LIN {X 0,Y 467.641,Z 718.232,A -85,B 0,C 180,E1 -7755.695,E2 -7755.695} C_VEL
LIN {X 0,Y 467.624,Z 718.234,A -85,B 0,C 180,E1 -7759.308,E2 -7759.308} C_VEL
LIN {X 0,Y 467.537,Z 718.247,A -85,B 0,C 180,E1 -7762.074,E2 -7762.074} C_VEL
LIN {X 0,Y 467.557,Z 718.246,A -85,B 0,C 180,E1 -7764.89,E2 -7764.89} C_VEL
LIN {X 0,Y 467.58,Z 718.239,A -85,B 0,C 180,E1 -7767.772,E2 -7767.772} C_VEL
LIN {X 0,Y 467.569,Z 718.244,A -85,B 0,C 180,E1 -7771.045,E2 -7771.045} C_VEL
LIN {X 0,Y 467.578,Z 718.242,A -85,B 0,C 180,E1 -7774.24,E2 -7774.24} C_VEL
LIN {X 0,Y 467.537,Z 718.248,A -85,B 0,C 180,E1 -7777.184,E2 -7777.184} C_VEL
LIN {X 0,Y 467.558,Z 718.244,A -85,B 0,C 180,E1 -7780.267,E2 -7780.267} C_VEL
LIN {X 0,Y 467.546,Z 718.243,A -85,B 0,C 180,E1 -7783.746,E2 -7783.746} C_VEL
LIN {X 0,Y 467.546,Z 718.244,A -85,B 0,C 180,E1 -7786.254,E2 -7786.254} C_VEL
LIN {X 0,Y 467.558,Z 718.242,A -85,B 0,C 180,E1 -7789.733,E2 -7789.733} C_VEL
LIN {X 0,Y 467.519,Z 718.25,A -85,B 0,C 180,E1 -7792.819,E2 -7792.819} C_VEL
LIN {X 0,Y 467.566,Z 718.242,A -85,B 0,C 180,E1 -7795.762,E2 -7795.762} C_VEL
LIN {X 0,Y 467.537,Z 718.248,A -85,B 0,C 180,E1 -7798.962,E2 -7798.962} C_VEL
LIN {X 0,Y 467.543,Z 718.244,A -85,B 0,C 180,E1 -7802.226,E2 -7802.226} C_VEL
LIN {X 0,Y 467.551,Z 718.246,A -85,B 0,C 180,E1 -7805.11,E2 -7805.11} C_VEL
LIN {X 0,Y 467.534,Z 718.246,A -85,B 0,C 180,E1 -7807.926,E2 -7807.926} C_VEL
LIN {X 0,Y 467.623,Z 718.234,A -85,B 0,C 180,E1 -7810.692,E2 -7810.692} C_VEL
LIN {X 0,Y 467.64,Z 718.231,A -85,B 0,C 180,E1 -7814.305,E2 -7814.305} C_VEL
LIN {X 0,Y 467.591,Z 718.24,A -85,B 0,C 180,E1 -7815.403,E2 -7815.403} C_VEL
LIN {X 0,Y 466.918,Z 718.323,A -85,B 0,C 180,E1 -7816.122,E2 -7816.122} C_VEL
LIN {X 0,Y 464.072,Z 718.68,A -85,B 0,C 180,E1 -7817.291,E2 -7817.291} C_VEL
LIN {X 0,Y 461.669,Z 718.976,A -85,B 0,C 180,E1 -7818.233,E2 -7818.233} C_VEL
LIN {X 0,Y 460.636,Z 719.106,A -85,B 0,C 180,E1 -7818.961,E2 -7818.961} C_VEL
LIN {X 0,Y 460.55,Z 719.116,A -85,B 0,C 180,E1 -7819.207,E2 -7819.207} C_VEL
LIN {X 0,Y 460.666,Z 719.1,A -85,B 0,C 180,E1 -7822.594,E2 -7822.594} C_VEL
LIN {X 0,Y 460.676,Z 719.099,A -85,B 0,C 180,E1 -7824.748,E2 -7824.748} C_VEL
LIN {X 0,Y 460.758,Z 719.093,A -85,B 0,C 180,E1 -7827.377,E2 -7827.377} C_VEL
LIN {X 0,Y 460.822,Z 719.082,A -85,B 0,C 180,E1 -7830,E2 -7830} C_VEL
LIN {X 0,Y 460.76,Z 719.088,A -85,B 0,C 180,E1 -7832.623,E2 -7832.623} C_VEL
LIN {X 0,Y 460.672,Z 719.101,A -85,B 0,C 180,E1 -7836.131,E2 -7836.131} C_VEL
LIN {X 0,Y 460.613,Z 719.106,A -85,B 0,C 180,E1 -7838.777,E2 -7838.777} C_VEL
LIN {X 0,Y 460.618,Z 719.107,A -85,B 0,C 180,E1 -7842.445,E2 -7842.445} C_VEL
LIN {X 0,Y 460.604,Z 719.112,A -85,B 0,C 180,E1 -7845.998,E2 -7845.998} C_VEL
LIN {X 0,Y 460.571,Z 719.114,A -85,B 0,C 180,E1 -7849.616,E2 -7849.616} C_VEL
LIN {X 0,Y 460.514,Z 719.12,A -85,B 0,C 180,E1 -7852.429,E2 -7852.429} C_VEL
LIN {X 0,Y 460.539,Z 719.118,A -85,B 0,C 180,E1 -7855.793,E2 -7855.793} C_VEL
LIN {X 0,Y 460.529,Z 719.121,A -85,B 0,C 180,E1 -7858.235,E2 -7858.235} C_VEL
LIN {X 0,Y 460.524,Z 719.116,A -85,B 0,C 180,E1 -7861.283,E2 -7861.283} C_VEL
LIN {X 0,Y 460.527,Z 719.12,A -85,B 0,C 180,E1 -7864.504,E2 -7864.504} C_VEL
LIN {X 0,Y 460.505,Z 719.119,A -85,B 0,C 180,E1 -7867.623,E2 -7867.623} C_VEL
LIN {X 0,Y 460.543,Z 719.12,A -85,B 0,C 180,E1 -7870.269,E2 -7870.269} C_VEL
LIN {X 0,Y 460.5,Z 719.118,A -85,B 0,C 180,E1 -7873.376,E2 -7873.376} C_VEL
LIN {X 0,Y 460.503,Z 719.125,A -85,B 0,C 180,E1 -7876.625,E2 -7876.625} C_VEL
LIN {X 0,Y 460.551,Z 719.173,A -85,B 0,C 180,E1 -7877.312,E2 -7877.312} C_VEL
LIN {X 0,Y 463.389,Z 730.051,A -85,B 0,C 180,E1 -7878.002,E2 -7878.002} C_VEL
LIN {X 0,Y 462.958,Z 741.918,A -85,B 0,C 180,E1 -7878.817,E2 -7878.817} C_VEL
LIN {X 0,Y 462.516,Z 752.947,A -85,B 0,C 180,E1 -7879.774,E2 -7879.774} C_VEL
LIN {X 0,Y 462.135,Z 762.944,A -85,B 0,C 180,E1 -7880.859,E2 -7880.859} C_VEL
LIN {X 0,Y 461.733,Z 771.018,A -85,B 0,C 180,E1 -7881.926,E2 -7881.926} C_VEL
LIN {X 0,Y 461.288,Z 779.332,A -85,B 0,C 180,E1 -7883.273,E2 -7883.273} C_VEL
LIN {X 0,Y 460.993,Z 785.888,A -85,B 0,C 180,E1 -7884.597,E2 -7884.597} C_VEL
LIN {X 0,Y 460.671,Z 791.9,A -85,B 0,C 180,E1 -7886.162,E2 -7886.162} C_VEL
LIN {X 0,Y 460.529,Z 796.315,A -85,B 0,C 180,E1 -7887.715,E2 -7887.715} C_VEL
LIN {X 0,Y 460.431,Z 798.454,A -85,B 0,C 180,E1 -7888.736,E2 -7888.736} C_VEL
LIN {X 0,Y 460.318,Z 800.811,A -85,B 0,C 180,E1 -7890.489,E2 -7890.489} C_VEL
LIN {X 0,Y 460.262,Z 801.563,A -85,B 0,C 180,E1 -7892.331,E2 -7892.331} C_VEL
LIN {X 0,Y 460.381,Z 800.51,A -85,B 0,C 180,E1 -7894.247,E2 -7894.247} C_VEL
LIN {X 0,Y 460.545,Z 798.474,A -85,B 0,C 180,E1 -7895.668,E2 -7895.668} C_VEL
LIN {X 0,Y 460.737,Z 795.274,A -85,B 0,C 180,E1 -7897.109,E2 -7897.109} C_VEL
LIN {X 0,Y 460.938,Z 790.895,A -85,B 0,C 180,E1 -7898.535,E2 -7898.535} C_VEL
LIN {X 0,Y 461.317,Z 785.168,A -85,B 0,C 180,E1 -7899.954,E2 -7899.954} C_VEL
LIN {X 0,Y 461.703,Z 777.905,A -85,B 0,C 180,E1 -7901.357,E2 -7901.357} C_VEL
LIN {X 0,Y 462.128,Z 770.414,A -85,B 0,C 180,E1 -7902.521,E2 -7902.521} C_VEL
LIN {X 0,Y 462.617,Z 761.045,A -85,B 0,C 180,E1 -7903.706,E2 -7903.706} C_VEL
LIN {X 0,Y 463.073,Z 751.217,A -85,B 0,C 180,E1 -7904.71,E2 -7904.71} C_VEL
LIN {X 0,Y 463.437,Z 740.075,A -85,B 0,C 180,E1 -7905.621,E2 -7905.621} C_VEL
LIN {X 0,Y 463.673,Z 729.937,A -85,B 0,C 180,E1 -7906.283,E2 -7906.283} C_VEL
LIN {X 0,Y 460.563,Z 719.117,A -85,B 0,C 180,E1 -7906.993,E2 -7906.993} C_VEL
LIN {X 0,Y 460.578,Z 719.118,A -85,B 0,C 180,E1 -7909.449,E2 -7909.449} C_VEL
LIN {X 0,Y 460.669,Z 719.099,A -85,B 0,C 180,E1 -7912.591,E2 -7912.591} C_VEL
LIN {X 0,Y 460.689,Z 719.096,A -85,B 0,C 180,E1 -7914.748,E2 -7914.748} C_VEL
LIN {X 0,Y 460.795,Z 719.088,A -85,B 0,C 180,E1 -7917.377,E2 -7917.377} C_VEL
LIN {X 0,Y 460.854,Z 719.081,A -85,B 0,C 180,E1 -7920,E2 -7920} C_VEL
LIN {X 0,Y 460.796,Z 719.08,A -85,B 0,C 180,E1 -7922.622,E2 -7922.622} C_VEL
LIN {X 0,Y 460.706,Z 719.096,A -85,B 0,C 180,E1 -7926.13,E2 -7926.13} C_VEL
LIN {X 0,Y 460.623,Z 719.1,A -85,B 0,C 180,E1 -7928.776,E2 -7928.776} C_VEL
LIN {X 0,Y 460.618,Z 719.108,A -85,B 0,C 180,E1 -7932.445,E2 -7932.445} C_VEL
LIN {X 0,Y 460.604,Z 719.109,A -85,B 0,C 180,E1 -7935.997,E2 -7935.997} C_VEL
LIN {X 0,Y 460.572,Z 719.112,A -85,B 0,C 180,E1 -7939.615,E2 -7939.615} C_VEL
LIN {X 0,Y 460.514,Z 719.123,A -85,B 0,C 180,E1 -7942.428,E2 -7942.428} C_VEL
LIN {X 0,Y 460.556,Z 719.115,A -85,B 0,C 180,E1 -7945.798,E2 -7945.798} C_VEL
LIN {X 0,Y 460.556,Z 719.119,A -85,B 0,C 180,E1 -7948.233,E2 -7948.233} C_VEL
LIN {X 0,Y 460.525,Z 719.116,A -85,B 0,C 180,E1 -7951.283,E2 -7951.283} C_VEL
LIN {X 0,Y 460.535,Z 719.122,A -85,B 0,C 180,E1 -7954.505,E2 -7954.505} C_VEL
LIN {X 0,Y 460.504,Z 719.123,A -85,B 0,C 180,E1 -7957.623,E2 -7957.623} C_VEL
LIN {X 0,Y 460.545,Z 719.122,A -85,B 0,C 180,E1 -7960.269,E2 -7960.269} C_VEL
LIN {X 0,Y 460.503,Z 719.123,A -85,B 0,C 180,E1 -7963.375,E2 -7963.375} C_VEL
LIN {X 0,Y 460.503,Z 719.126,A -85,B 0,C 180,E1 -7966.625,E2 -7966.625} C_VEL
LIN {X 0,Y 460.569,Z 719.225,A -85,B 0,C 180,E1 -7969.186,E2 -7969.186} C_VEL
LIN {X 0,Y 462.284,Z 727.914,A -85,B 0,C 180,E1 -7971.868,E2 -7971.868} C_VEL
LIN {X 0,Y 463.24,Z 733.679,A -85,B 0,C 180,E1 -7973.522,E2 -7973.522} C_VEL
LIN {X 0,Y 462.632,Z 745.802,A -85,B 0,C 180,E1 -7976.671,E2 -7976.671} C_VEL
LIN {X 0,Y 462.154,Z 756.733,A -85,B 0,C 180,E1 -7979.373,E2 -7979.373} C_VEL
LIN {X 0,Y 461.717,Z 769.456,A -85,B 0,C 180,E1 -7982.401,E2 -7982.401} C_VEL
LIN {X 0,Y 461.325,Z 782.735,A -85,B 0,C 180,E1 -7985.472,E2 -7985.472} C_VEL
LIN {X 0,Y 460.896,Z 798.404,A -85,B 0,C 180,E1 -7989.001,E2 -7989.001} C_VEL
LIN {X 0,Y 460.603,Z 813.029,A -85,B 0,C 180,E1 -7992.232,E2 -7992.232} C_VEL
LIN {X 0,Y 460.409,Z 822.488,A -85,B 0,C 180,E1 -7994.308,E2 -7994.308} C_VEL
LIN {X 0,Y 461.762,Z 838.292,A -85,B 0,C 180,E1 -7994.765,E2 -7994.765} C_VEL
LIN {X 0,Y 462.945,Z 847.629,A -85,B 0,C 180,E1 -7995.156,E2 -7995.156} C_VEL
LIN {X 0,Y 462.383,Z 860.861,A -85,B 0,C 180,E1 -7995.813,E2 -7995.813} C_VEL
LIN {X 0,Y 461.826,Z 872.507,A -85,B 0,C 180,E1 -7996.581,E2 -7996.581} C_VEL
LIN {X 0,Y 461.386,Z 884.01,A -85,B 0,C 180,E1 -7997.54,E2 -7997.54} C_VEL
LIN {X 0,Y 460.965,Z 894.018,A -85,B 0,C 180,E1 -7998.568,E2 -7998.568} C_VEL
LIN {X 0,Y 460.509,Z 902.816,A -85,B 0,C 180,E1 -7999.67,E2 -7999.67} C_VEL
LIN {X 0,Y 460.187,Z 911.411,A -85,B 0,C 180,E1 -8000.994,E2 -8000.994} C_VEL
LIN {X 0,Y 459.999,Z 918.373,A -85,B 0,C 180,E1 -8002.317,E2 -8002.317} C_VEL
LIN {X 0,Y 459.921,Z 924.781,A -85,B 0,C 180,E1 -8003.859,E2 -8003.859} C_VEL
LIN {X 0,Y 459.81,Z 928.937,A -85,B 0,C 180,E1 -8005.178,E2 -8005.178} C_VEL
LIN {X 0,Y 459.806,Z 932.028,A -85,B 0,C 180,E1 -8006.495,E2 -8006.495} C_VEL
LIN {X 0,Y 459.772,Z 933.497,A -85,B 0,C 180,E1 -8007.372,E2 -8007.372} C_VEL
LIN {X 0,Y 459.759,Z 934.556,A -85,B 0,C 180,E1 -8008.248,E2 -8008.248} C_VEL
LIN {X 0,Y 459.72,Z 935.213,A -85,B 0,C 180,E1 -8009.124,E2 -8009.124} C_VEL
LIN {X 0,Y 459.708,Z 935.461,A -85,B 0,C 180,E1 -8010,E2 -8010} C_VEL
LIN {X 0,Y 459.714,Z 935.257,A -85,B 0,C 180,E1 -8010.876,E2 -8010.876} C_VEL
LIN {X 0,Y 459.747,Z 934.654,A -85,B 0,C 180,E1 -8011.752,E2 -8011.752} C_VEL
LIN {X 0,Y 459.756,Z 933.651,A -85,B 0,C 180,E1 -8012.628,E2 -8012.628} C_VEL
LIN {X 0,Y 459.805,Z 932.229,A -85,B 0,C 180,E1 -8013.505,E2 -8013.505} C_VEL
LIN {X 0,Y 459.792,Z 929.22,A -85,B 0,C 180,E1 -8014.822,E2 -8014.822} C_VEL
LIN {X 0,Y 459.872,Z 925.148,A -85,B 0,C 180,E1 -8016.141,E2 -8016.141} C_VEL
LIN {X 0,Y 459.975,Z 918.865,A -85,B 0,C 180,E1 -8017.683,E2 -8017.683} C_VEL
LIN {X 0,Y 460.165,Z 912.028,A -85,B 0,C 180,E1 -8019.006,E2 -8019.006} C_VEL
LIN {X 0,Y 460.498,Z 903.571,A -85,B 0,C 180,E1 -8020.33,E2 -8020.33} C_VEL
LIN {X 0,Y 460.936,Z 894.899,A -85,B 0,C 180,E1 -8021.433,E2 -8021.433} C_VEL
LIN {X 0,Y 461.454,Z 884.841,A -85,B 0,C 180,E1 -8022.477,E2 -8022.477} C_VEL
LIN {X 0,Y 461.877,Z 873.701,A -85,B 0,C 180,E1 -8023.418,E2 -8023.418} C_VEL
LIN {X 0,Y 462.401,Z 862.191,A -85,B 0,C 180,E1 -8024.187,E2 -8024.187} C_VEL
LIN {X 0,Y 462.955,Z 849.085,A -85,B 0,C 180,E1 -8024.843,E2 -8024.843} C_VEL
LIN {X 0,Y 462.52,Z 843.463,A -85,B 0,C 180,E1 -8025.083,E2 -8025.083} C_VEL
LIN {X 0,Y 461.092,Z 830.929,A -85,B 0,C 180,E1 -8025.513,E2 -8025.513} C_VEL
LIN {X 0,Y 460.41,Z 824.173,A -85,B 0,C 180,E1 -8025.692,E2 -8025.692} C_VEL
LIN {X 0,Y 460.724,Z 810.998,A -85,B 0,C 180,E1 -8028.683,E2 -8028.683} C_VEL
LIN {X 0,Y 461.159,Z 796.773,A -85,B 0,C 180,E1 -8031.952,E2 -8031.952} C_VEL
LIN {X 0,Y 461.63,Z 783.77,A -85,B 0,C 180,E1 -8034.991,E2 -8034.991} C_VEL
LIN {X 0,Y 462.165,Z 771.673,A -85,B 0,C 180,E1 -8037.874,E2 -8037.874} C_VEL
LIN {X 0,Y 462.764,Z 758.519,A -85,B 0,C 180,E1 -8041.088,E2 -8041.088} C_VEL
LIN {X 0,Y 463.449,Z 746.382,A -85,B 0,C 180,E1 -8044.131,E2 -8044.131} C_VEL
LIN {X 0,Y 463.948,Z 736.881,A -85,B 0,C 180,E1 -8046.596,E2 -8046.596} C_VEL
LIN {X 0,Y 463.061,Z 731.333,A -85,B 0,C 180,E1 -8048.148,E2 -8048.148} C_VEL
LIN {X 0,Y 460.655,Z 719.583,A -85,B 0,C 180,E1 -8051.62,E2 -8051.62} C_VEL
LIN {X 0,Y 460.543,Z 719.12,A -85,B 0,C 180,E1 -8051.857,E2 -8051.857} C_VEL
LIN {X 0,Y 460.519,Z 719.122,A -85,B 0,C 180,E1 -8055.412,E2 -8055.412} C_VEL
LIN {X 0,Y 460.534,Z 719.117,A -85,B 0,C 180,E1 -8058.397,E2 -8058.397} C_VEL
LIN {X 0,Y 460.529,Z 719.121,A -85,B 0,C 180,E1 -8061.267,E2 -8061.267} C_VEL
LIN {X 0,Y 460.513,Z 719.117,A -85,B 0,C 180,E1 -8064.554,E2 -8064.554} C_VEL
LIN {X 0,Y 460.534,Z 719.121,A -85,B 0,C 180,E1 -8067.716,E2 -8067.716} C_VEL
LIN {X 0,Y 460.542,Z 719.114,A -85,B 0,C 180,E1 -8070.769,E2 -8070.769} C_VEL
LIN {X 0,Y 460.558,Z 719.119,A -85,B 0,C 180,E1 -8073.734,E2 -8073.734} C_VEL
LIN {X 0,Y 460.547,Z 719.114,A -85,B 0,C 180,E1 -8076.624,E2 -8076.624} C_VEL
LIN {X 0,Y 460.553,Z 719.115,A -85,B 0,C 180,E1 -8079.453,E2 -8079.453} C_VEL
LIN {X 0,Y 460.553,Z 719.116,A -85,B 0,C 180,E1 -8082.23,E2 -8082.23} C_VEL
LIN {X 0,Y 460.568,Z 719.112,A -85,B 0,C 180,E1 -8084.965,E2 -8084.965} C_VEL
LIN {X 0,Y 460.613,Z 719.107,A -85,B 0,C 180,E1 -8088.559,E2 -8088.559} C_VEL
LIN {X 0,Y 460.698,Z 719.101,A -85,B 0,C 180,E1 -8092.109,E2 -8092.109} C_VEL
LIN {X 0,Y 460.697,Z 719.096,A -85,B 0,C 180,E1 -8094.748,E2 -8094.748} C_VEL
LIN {X 0,Y 460.791,Z 719.085,A -85,B 0,C 180,E1 -8097.378,E2 -8097.378} C_VEL
LIN {X 0,Y 460.853,Z 719.079,A -85,B 0,C 180,E1 -8100,E2 -8100} C_VEL
LIN {X 0,Y 460.794,Z 719.087,A -85,B 0,C 180,E1 -8102.623,E2 -8102.623} C_VEL
LIN {X 0,Y 460.684,Z 719.1,A -85,B 0,C 180,E1 -8106.13,E2 -8106.13} C_VEL
LIN {X 0,Y 460.622,Z 719.108,A -85,B 0,C 180,E1 -8108.776,E2 -8108.776} C_VEL
LIN {X 0,Y 460.616,Z 719.11,A -85,B 0,C 180,E1 -8112.445,E2 -8112.445} C_VEL
LIN {X 0,Y 460.603,Z 719.11,A -85,B 0,C 180,E1 -8115.998,E2 -8115.998} C_VEL
LIN {X 0,Y 460.57,Z 719.112,A -85,B 0,C 180,E1 -8119.616,E2 -8119.616} C_VEL
LIN {X 0,Y 460.513,Z 719.122,A -85,B 0,C 180,E1 -8122.429,E2 -8122.429} C_VEL
LIN {X 0,Y 460.534,Z 719.117,A -85,B 0,C 180,E1 -8125.793,E2 -8125.793} C_VEL
LIN {X 0,Y 460.527,Z 719.12,A -85,B 0,C 180,E1 -8128.235,E2 -8128.235} C_VEL
LIN {X 0,Y 460.522,Z 719.12,A -85,B 0,C 180,E1 -8131.283,E2 -8131.283} C_VEL
LIN {X 0,Y 460.523,Z 719.121,A -85,B 0,C 180,E1 -8134.504,E2 -8134.504} C_VEL
LIN {X 0,Y 460.494,Z 719.122,A -85,B 0,C 180,E1 -8137.624,E2 -8137.624} C_VEL
LIN {X 0,Y 460.516,Z 719.122,A -85,B 0,C 180,E1 -8141.013,E2 -8141.013} C_VEL
LIN {X 0,Y 460.513,Z 719.123,A -85,B 0,C 180,E1 -8144.589,E2 -8144.589} C_VEL
LIN {X 0,Y 460.477,Z 719.124,A -85,B 0,C 180,E1 -8147.813,E2 -8147.813} C_VEL
LIN {X 0,Y 460.511,Z 719.12,A -85,B 0,C 180,E1 -8150.135,E2 -8150.135} C_VEL
LIN {X 0,Y 460.462,Z 719.129,A -85,B 0,C 180,E1 -8153.469,E2 -8153.469} C_VEL
LIN {X 0,Y 460.502,Z 719.124,A -85,B 0,C 180,E1 -8156.673,E2 -8156.673} C_VEL
LIN {X 0,Y 460.495,Z 719.123,A -85,B 0,C 180,E1 -8159.759,E2 -8159.759} C_VEL
LIN {X 0,Y 460.486,Z 719.125,A -85,B 0,C 180,E1 -8162.751,E2 -8162.751} C_VEL
LIN {X 0,Y 460.515,Z 719.122,A -85,B 0,C 180,E1 -8165.666,E2 -8165.666} C_VEL
LIN {X 0,Y 460.525,Z 719.119,A -85,B 0,C 180,E1 -8168.578,E2 -8168.578} C_VEL
LIN {X 0,Y 460.587,Z 719.113,A -85,B 0,C 180,E1 -8171.311,E2 -8171.311} C_VEL
LIN {X 0,Y 460.589,Z 719.111,A -85,B 0,C 180,E1 -8174.058,E2 -8174.058} C_VEL
LIN {X 0,Y 460.606,Z 719.11,A -85,B 0,C 180,E1 -8177.666,E2 -8177.666} C_VEL
LIN {X 0,Y 460.55,Z 719.116,A -85,B 0,C 180,E1 -8179.207,E2 -8179.207} C_VEL
LIN {X 0,Y 459.885,Z 719.203,A -85,B 0,C 180,E1 -8179.937,E2 -8179.937} C_VEL
LIN {X 0,Y 457.054,Z 719.557,A -85,B 0,C 180,E1 -8181.123,E2 -8181.123} C_VEL
LIN {X 0,Y 454.672,Z 719.851,A -85,B 0,C 180,E1 -8182.08,E2 -8182.08} C_VEL
LIN {X 0,Y 453.663,Z 719.973,A -85,B 0,C 180,E1 -8182.818,E2 -8182.818} C_VEL
LIN {X 0,Y 453.588,Z 719.982,A -85,B 0,C 180,E1 -8183.068,E2 -8183.068} C_VEL
LIN {X 0,Y 453.649,Z 719.974,A -85,B 0,C 180,E1 -8184.667,E2 -8184.667} C_VEL
LIN {X 0,Y 453.689,Z 719.971,A -85,B 0,C 180,E1 -8188.225,E2 -8188.225} C_VEL
LIN {X 0,Y 453.771,Z 719.961,A -85,B 0,C 180,E1 -8190,E2 -8190} C_VEL
LIN {X 0,Y 453.707,Z 719.967,A -85,B 0,C 180,E1 -8192.664,E2 -8192.664} C_VEL
LIN {X 0,Y 453.64,Z 719.976,A -85,B 0,C 180,E1 -8196.226,E2 -8196.226} C_VEL
LIN {X 0,Y 453.581,Z 719.982,A -85,B 0,C 180,E1 -8198.914,E2 -8198.914} C_VEL
LIN {X 0,Y 453.568,Z 719.985,A -85,B 0,C 180,E1 -8202.529,E2 -8202.529} C_VEL
LIN {X 0,Y 453.548,Z 719.989,A -85,B 0,C 180,E1 -8206.196,E2 -8206.196} C_VEL
LIN {X 0,Y 453.52,Z 719.989,A -85,B 0,C 180,E1 -8209.039,E2 -8209.039} C_VEL
LIN {X 0,Y 453.48,Z 719.999,A -85,B 0,C 180,E1 -8211.836,E2 -8211.836} C_VEL
LIN {X 0,Y 453.494,Z 719.993,A -85,B 0,C 180,E1 -8214.736,E2 -8214.736} C_VEL
LIN {X 0,Y 453.509,Z 719.996,A -85,B 0,C 180,E1 -8217.953,E2 -8217.953} C_VEL
LIN {X 0,Y 453.479,Z 719.995,A -85,B 0,C 180,E1 -8220.76,E2 -8220.76} C_VEL
LIN {X 0,Y 453.472,Z 719.998,A -85,B 0,C 180,E1 -8223.913,E2 -8223.913} C_VEL
LIN {X 0,Y 453.456,Z 719.997,A -85,B 0,C 180,E1 -8227.19,E2 -8227.19} C_VEL
LIN {X 0,Y 453.487,Z 719.992,A -85,B 0,C 180,E1 -8229.45,E2 -8229.45} C_VEL
LIN {X 0,Y 453.48,Z 719.995,A -85,B 0,C 180,E1 -8231.935,E2 -8231.935} C_VEL
LIN {X 0,Y 453.488,Z 719.994,A -85,B 0,C 180,E1 -8235.471,E2 -8235.471} C_VEL
LIN {X 0,Y 453.479,Z 720.021,A -85,B 0,C 180,E1 -8237.09,E2 -8237.09} C_VEL
LIN {X 0,Y 456.413,Z 730.363,A -85,B 0,C 180,E1 -8237.761,E2 -8237.761} C_VEL
LIN {X 0,Y 456.11,Z 742.427,A -85,B 0,C 180,E1 -8238.598,E2 -8238.598} C_VEL
LIN {X 0,Y 455.624,Z 754.065,A -85,B 0,C 180,E1 -8239.62,E2 -8239.62} C_VEL
LIN {X 0,Y 455.197,Z 764.082,A -85,B 0,C 180,E1 -8240.727,E2 -8240.727} C_VEL
LIN {X 0,Y 454.724,Z 773.541,A -85,B 0,C 180,E1 -8242.021,E2 -8242.021} C_VEL
LIN {X 0,Y 454.312,Z 781.006,A -85,B 0,C 180,E1 -8243.28,E2 -8243.28} C_VEL
LIN {X 0,Y 454.013,Z 786.956,A -85,B 0,C 180,E1 -8244.515,E2 -8244.515} C_VEL
LIN {X 0,Y 453.681,Z 792.959,A -85,B 0,C 180,E1 -8246.104,E2 -8246.104} C_VEL
LIN {X 0,Y 453.523,Z 797.377,A -85,B 0,C 180,E1 -8247.681,E2 -8247.681} C_VEL
LIN {X 0,Y 453.352,Z 800.377,A -85,B 0,C 180,E1 -8249.231,E2 -8249.231} C_VEL
LIN {X 0,Y 453.296,Z 801.627,A -85,B 0,C 180,E1 -8250.255,E2 -8250.255} C_VEL
LIN {X 0,Y 453.27,Z 802.399,A -85,B 0,C 180,E1 -8251.271,E2 -8251.271} C_VEL
LIN {X 0,Y 453.247,Z 802.612,A -85,B 0,C 180,E1 -8252.278,E2 -8252.278} C_VEL
LIN {X 0,Y 453.346,Z 801.806,A -85,B 0,C 180,E1 -8254.047,E2 -8254.047} C_VEL
LIN {X 0,Y 453.486,Z 800.306,A -85,B 0,C 180,E1 -8255.264,E2 -8255.264} C_VEL
LIN {X 0,Y 453.681,Z 797.488,A -85,B 0,C 180,E1 -8256.732,E2 -8256.732} C_VEL
LIN {X 0,Y 453.943,Z 793.243,A -85,B 0,C 180,E1 -8258.269,E2 -8258.269} C_VEL
LIN {X 0,Y 454.321,Z 787.177,A -85,B 0,C 180,E1 -8259.867,E2 -8259.867} C_VEL
LIN {X 0,Y 454.748,Z 780.199,A -85,B 0,C 180,E1 -8261.295,E2 -8261.295} C_VEL
LIN {X 0,Y 455.172,Z 772.999,A -85,B 0,C 180,E1 -8262.477,E2 -8262.477} C_VEL
LIN {X 0,Y 455.689,Z 763.798,A -85,B 0,C 180,E1 -8263.698,E2 -8263.698} C_VEL
LIN {X 0,Y 456.159,Z 753.374,A -85,B 0,C 180,E1 -8264.816,E2 -8264.816} C_VEL
LIN {X 0,Y 456.64,Z 742.436,A -85,B 0,C 180,E1 -8265.744,E2 -8265.744} C_VEL
LIN {X 0,Y 456.937,Z 732.263,A -85,B 0,C 180,E1 -8266.435,E2 -8266.435} C_VEL
LIN {X 0,Y 454.255,Z 722.511,A -85,B 0,C 180,E1 -8267.087,E2 -8267.087} C_VEL
LIN {X 0,Y 453.556,Z 719.991,A -85,B 0,C 180,E1 -8267.243,E2 -8267.243} C_VEL
LIN {X 0,Y 453.574,Z 719.987,A -85,B 0,C 180,E1 -8270.186,E2 -8270.186} C_VEL
LIN {X 0,Y 453.59,Z 719.981,A -85,B 0,C 180,E1 -8272.88,E2 -8272.88} C_VEL
LIN {X 0,Y 453.661,Z 719.971,A -85,B 0,C 180,E1 -8274.667,E2 -8274.667} C_VEL
LIN {X 0,Y 453.739,Z 719.966,A -85,B 0,C 180,E1 -8277.337,E2 -8277.337} C_VEL
LIN {X 0,Y 453.824,Z 719.956,A -85,B 0,C 180,E1 -8280,E2 -8280} C_VEL
LIN {X 0,Y 453.74,Z 719.959,A -85,B 0,C 180,E1 -8282.663,E2 -8282.663} C_VEL
LIN {X 0,Y 453.673,Z 719.973,A -85,B 0,C 180,E1 -8286.225,E2 -8286.225} C_VEL
LIN {X 0,Y 453.589,Z 719.976,A -85,B 0,C 180,E1 -8288.913,E2 -8288.913} C_VEL
LIN {X 0,Y 453.568,Z 719.985,A -85,B 0,C 180,E1 -8292.529,E2 -8292.529} C_VEL
LIN {X 0,Y 453.548,Z 719.991,A -85,B 0,C 180,E1 -8296.196,E2 -8296.196} C_VEL
LIN {X 0,Y 453.521,Z 719.989,A -85,B 0,C 180,E1 -8299.039,E2 -8299.039} C_VEL
LIN {X 0,Y 453.48,Z 719.994,A -85,B 0,C 180,E1 -8301.836,E2 -8301.836} C_VEL
LIN {X 0,Y 453.504,Z 719.994,A -85,B 0,C 180,E1 -8304.735,E2 -8304.735} C_VEL
LIN {X 0,Y 453.536,Z 719.991,A -85,B 0,C 180,E1 -8307.959,E2 -8307.959} C_VEL
LIN {X 0,Y 453.469,Z 719.995,A -85,B 0,C 180,E1 -8311.525,E2 -8311.525} C_VEL
LIN {X 0,Y 453.491,Z 719.997,A -85,B 0,C 180,E1 -8314.777,E2 -8314.777} C_VEL
LIN {X 0,Y 453.468,Z 720.005,A -85,B 0,C 180,E1 -8318.311,E2 -8318.311} C_VEL
LIN {X 0,Y 453.497,Z 720,A -85,B 0,C 180,E1 -8320.609,E2 -8320.609} C_VEL
LIN {X 0,Y 453.459,Z 720.002,A -85,B 0,C 180,E1 -8323.244,E2 -8323.244} C_VEL
LIN {X 0,Y 453.469,Z 719.999,A -85,B 0,C 180,E1 -8325.779,E2 -8325.779} C_VEL
LIN {X 0,Y 453.522,Z 720.124,A -85,B 0,C 180,E1 -8328.854,E2 -8328.854} C_VEL
LIN {X 0,Y 455.244,Z 728.714,A -85,B 0,C 180,E1 -8331.583,E2 -8331.583} C_VEL
LIN {X 0,Y 456.191,Z 734.289,A -85,B 0,C 180,E1 -8333.236,E2 -8333.236} C_VEL
LIN {X 0,Y 455.937,Z 741.67,A -85,B 0,C 180,E1 -8335.226,E2 -8335.226} C_VEL
LIN {X 0,Y 455.305,Z 754.831,A -85,B 0,C 180,E1 -8338.603,E2 -8338.603} C_VEL
LIN {X 0,Y 454.718,Z 768.985,A -85,B 0,C 180,E1 -8342.062,E2 -8342.062} C_VEL
LIN {X 0,Y 454.311,Z 781.714,A -85,B 0,C 180,E1 -8345.068,E2 -8345.068} C_VEL
LIN {X 0,Y 453.914,Z 795.67,A -85,B 0,C 180,E1 -8348.278,E2 -8348.278} C_VEL
LIN {X 0,Y 453.53,Z 811.891,A -85,B 0,C 180,E1 -8351.945,E2 -8351.945} C_VEL
LIN {X 0,Y 453.313,Z 821.353,A -85,B 0,C 180,E1 -8354.059,E2 -8354.059} C_VEL
LIN {X 0,Y 454.617,Z 836.529,A -85,B 0,C 180,E1 -8354.499,E2 -8354.499} C_VEL
LIN {X 0,Y 455.937,Z 849.07,A -85,B 0,C 180,E1 -8355.037,E2 -8355.037} C_VEL
LIN {X 0,Y 455.352,Z 861.5,A -85,B 0,C 180,E1 -8355.703,E2 -8355.703} C_VEL
LIN {X 0,Y 454.786,Z 872.78,A -85,B 0,C 180,E1 -8356.483,E2 -8356.483} C_VEL
LIN {X 0,Y 454.341,Z 882.583,A -85,B 0,C 180,E1 -8357.321,E2 -8357.321} C_VEL
LIN {X 0,Y 453.868,Z 892.835,A -85,B 0,C 180,E1 -8358.387,E2 -8358.387} C_VEL
LIN {X 0,Y 453.446,Z 901.666,A -85,B 0,C 180,E1 -8359.507,E2 -8359.507} C_VEL
LIN {X 0,Y 453.139,Z 910.293,A -85,B 0,C 180,E1 -8360.853,E2 -8360.853} C_VEL
LIN {X 0,Y 452.925,Z 917.273,A -85,B 0,C 180,E1 -8362.197,E2 -8362.197} C_VEL
LIN {X 0,Y 452.865,Z 923.706,A -85,B 0,C 180,E1 -8363.763,E2 -8363.763} C_VEL
LIN {X 0,Y 452.774,Z 927.883,A -85,B 0,C 180,E1 -8365.102,E2 -8365.102} C_VEL
LIN {X 0,Y 452.768,Z 930.989,A -85,B 0,C 180,E1 -8366.44,E2 -8366.44} C_VEL
LIN {X 0,Y 452.734,Z 932.466,A -85,B 0,C 180,E1 -8367.331,E2 -8367.331} C_VEL
LIN {X 0,Y 452.725,Z 933.537,A -85,B 0,C 180,E1 -8368.221,E2 -8368.221} C_VEL
LIN {X 0,Y 452.691,Z 934.2,A -85,B 0,C 180,E1 -8369.11,E2 -8369.11} C_VEL
LIN {X 0,Y 452.68,Z 934.454,A -85,B 0,C 180,E1 -8370,E2 -8370} C_VEL
LIN {X 0,Y 452.684,Z 934.253,A -85,B 0,C 180,E1 -8370.889,E2 -8370.889} C_VEL
LIN {X 0,Y 452.71,Z 933.657,A -85,B 0,C 180,E1 -8371.779,E2 -8371.779} C_VEL
LIN {X 0,Y 452.716,Z 932.655,A -85,B 0,C 180,E1 -8372.669,E2 -8372.669} C_VEL
LIN {X 0,Y 452.767,Z 931.236,A -85,B 0,C 180,E1 -8373.56,E2 -8373.56} C_VEL
LIN {X 0,Y 452.752,Z 928.228,A -85,B 0,C 180,E1 -8374.898,E2 -8374.898} C_VEL
LIN {X 0,Y 452.798,Z 924.152,A -85,B 0,C 180,E1 -8376.237,E2 -8376.237} C_VEL
LIN {X 0,Y 452.909,Z 917.869,A -85,B 0,C 180,E1 -8377.804,E2 -8377.804} C_VEL
LIN {X 0,Y 453.119,Z 911.033,A -85,B 0,C 180,E1 -8379.148,E2 -8379.148} C_VEL
LIN {X 0,Y 453.439,Z 902.567,A -85,B 0,C 180,E1 -8380.493,E2 -8380.493} C_VEL
LIN {X 0,Y 453.875,Z 893.886,A -85,B 0,C 180,E1 -8381.613,E2 -8381.613} C_VEL
LIN {X 0,Y 454.436,Z 884.13,A -85,B 0,C 180,E1 -8382.645,E2 -8382.645} C_VEL
LIN {X 0,Y 454.894,Z 872.692,A -85,B 0,C 180,E1 -8383.627,E2 -8383.627} C_VEL
LIN {X 0,Y 455.506,Z 861.186,A -85,B 0,C 180,E1 -8384.406,E2 -8384.406} C_VEL
LIN {X 0,Y 456.038,Z 848.083,A -85,B 0,C 180,E1 -8385.074,E2 -8385.074} C_VEL
LIN {X 0,Y 454.644,Z 835.797,A -85,B 0,C 180,E1 -8385.577,E2 -8385.577} C_VEL
LIN {X 0,Y 453.373,Z 823.286,A -85,B 0,C 180,E1 -8385.943,E2 -8385.943} C_VEL
LIN {X 0,Y 453.663,Z 810.143,A -85,B 0,C 180,E1 -8388.985,E2 -8388.985} C_VEL
LIN {X 0,Y 454.116,Z 797.083,A -85,B 0,C 180,E1 -8392.043,E2 -8392.043} C_VEL
LIN {X 0,Y 454.625,Z 783.999,A -85,B 0,C 180,E1 -8395.158,E2 -8395.158} C_VEL
LIN {X 0,Y 455.139,Z 772.406,A -85,B 0,C 180,E1 -8397.973,E2 -8397.973} C_VEL
LIN {X 0,Y 455.834,Z 758.813,A -85,B 0,C 180,E1 -8401.356,E2 -8401.356} C_VEL
LIN {X 0,Y 456.551,Z 746.701,A -85,B 0,C 180,E1 -8404.452,E2 -8404.452} C_VEL
LIN {X 0,Y 456.975,Z 737.484,A -85,B 0,C 180,E1 -8406.896,E2 -8406.896} C_VEL
LIN {X 0,Y 455.226,Z 728.603,A -85,B 0,C 180,E1 -8409.473,E2 -8409.473} C_VEL
LIN {X 0,Y 453.516,Z 719.994,A -85,B 0,C 180,E1 -8412.143,E2 -8412.143} C_VEL
LIN {X 0,Y 453.489,Z 719.998,A -85,B 0,C 180,E1 -8415.471,E2 -8415.471} C_VEL
LIN {X 0,Y 453.481,Z 719.996,A -85,B 0,C 180,E1 -8418.209,E2 -8418.209} C_VEL
LIN {X 0,Y 453.497,Z 719.993,A -85,B 0,C 180,E1 -8420.793,E2 -8420.793} C_VEL
LIN {X 0,Y 453.456,Z 719.999,A -85,B 0,C 180,E1 -8423.917,E2 -8423.917} C_VEL
LIN {X 0,Y 453.485,Z 719.995,A -85,B 0,C 180,E1 -8427.151,E2 -8427.151} C_VEL
LIN {X 0,Y 453.477,Z 719.995,A -85,B 0,C 180,E1 -8430.268,E2 -8430.268} C_VEL
LIN {X 0,Y 453.504,Z 719.993,A -85,B 0,C 180,E1 -8433.294,E2 -8433.294} C_VEL
LIN {X 0,Y 453.5,Z 719.994,A -85,B 0,C 180,E1 -8436.239,E2 -8436.239} C_VEL
LIN {X 0,Y 453.485,Z 719.995,A -85,B 0,C 180,E1 -8439.118,E2 -8439.118} C_VEL
LIN {X 0,Y 453.507,Z 719.998,A -85,B 0,C 180,E1 -8441.944,E2 -8441.944} C_VEL
LIN {X 0,Y 453.542,Z 719.987,A -85,B 0,C 180,E1 -8444.726,E2 -8444.726} C_VEL
LIN {X 0,Y 453.562,Z 719.987,A -85,B 0,C 180,E1 -8448.379,E2 -8448.379} C_VEL
LIN {X 0,Y 453.655,Z 719.977,A -85,B 0,C 180,E1 -8451.985,E2 -8451.985} C_VEL
LIN {X 0,Y 453.671,Z 719.972,A -85,B 0,C 180,E1 -8454.667,E2 -8454.667} C_VEL
LIN {X 0,Y 453.735,Z 719.964,A -85,B 0,C 180,E1 -8457.337,E2 -8457.337} C_VEL
LIN {X 0,Y 453.823,Z 719.955,A -85,B 0,C 180,E1 -8460,E2 -8460} C_VEL
LIN {X 0,Y 453.738,Z 719.965,A -85,B 0,C 180,E1 -8462.663,E2 -8462.663} C_VEL
LIN {X 0,Y 453.65,Z 719.977,A -85,B 0,C 180,E1 -8466.226,E2 -8466.226} C_VEL
LIN {X 0,Y 453.588,Z 719.983,A -85,B 0,C 180,E1 -8468.914,E2 -8468.914} C_VEL
LIN {X 0,Y 453.566,Z 719.989,A -85,B 0,C 180,E1 -8472.529,E2 -8472.529} C_VEL
LIN {X 0,Y 453.547,Z 719.989,A -85,B 0,C 180,E1 -8476.196,E2 -8476.196} C_VEL
LIN {X 0,Y 453.519,Z 719.992,A -85,B 0,C 180,E1 -8479.039,E2 -8479.039} C_VEL
LIN {X 0,Y 453.479,Z 719.997,A -85,B 0,C 180,E1 -8481.836,E2 -8481.836} C_VEL
LIN {X 0,Y 453.47,Z 720,A -85,B 0,C 180,E1 -8484.737,E2 -8484.737} C_VEL
LIN {X 0,Y 453.492,Z 719.995,A -85,B 0,C 180,E1 -8487.949,E2 -8487.949} C_VEL
LIN {X 0,Y 453.477,Z 719.998,A -85,B 0,C 180,E1 -8490.76,E2 -8490.76} C_VEL
LIN {X 0,Y 453.468,Z 719.998,A -85,B 0,C 180,E1 -8493.914,E2 -8493.914} C_VEL
LIN {X 0,Y 453.446,Z 720.003,A -85,B 0,C 180,E1 -8497.191,E2 -8497.191} C_VEL
LIN {X 0,Y 453.471,Z 719.999,A -85,B 0,C 180,E1 -8500.612,E2 -8500.612} C_VEL
LIN {X 0,Y 453.483,Z 719.999,A -85,B 0,C 180,E1 -8504.528,E2 -8504.528} C_VEL
LIN {X 0,Y 453.438,Z 720.001,A -85,B 0,C 180,E1 -8508.071,E2 -8508.071} C_VEL
LIN {X 0,Y 453.44,Z 720.003,A -85,B 0,C 180,E1 -8510.802,E2 -8510.802} C_VEL
LIN {X 0,Y 453.444,Z 720.001,A -85,B 0,C 180,E1 -8513.916,E2 -8513.916} C_VEL
LIN {X 0,Y 453.466,Z 720.001,A -85,B 0,C 180,E1 -8516.816,E2 -8516.816} C_VEL
LIN {X 0,Y 453.456,Z 719.999,A -85,B 0,C 180,E1 -8520.267,E2 -8520.267} C_VEL
LIN {X 0,Y 453.425,Z 720.005,A -85,B 0,C 180,E1 -8523.289,E2 -8523.289} C_VEL
LIN {X 0,Y 453.493,Z 719.994,A -85,B 0,C 180,E1 -8526.238,E2 -8526.238} C_VEL
LIN {X 0,Y 453.485,Z 719.999,A -85,B 0,C 180,E1 -8529.118,E2 -8529.118} C_VEL
LIN {X 0,Y 453.5,Z 719.995,A -85,B 0,C 180,E1 -8531.944,E2 -8531.944} C_VEL
LIN {X 0,Y 453.533,Z 719.99,A -85,B 0,C 180,E1 -8534.726,E2 -8534.726} C_VEL
LIN {X 0,Y 453.546,Z 719.987,A -85,B 0,C 180,E1 -8538.379,E2 -8538.379} C_VEL
LIN {X 0,Y 453.557,Z 719.988,A -85,B 0,C 180,E1 -8541.086,E2 -8541.086} C_VEL
LIN {X 0,Y 453.588,Z 719.982,A -85,B 0,C 180,E1 -8543.068,E2 -8543.068} C_VEL
LIN {X 0,Y 452.907,Z 720.069,A -85,B 0,C 180,E1 -8543.809,E2 -8543.809} C_VEL
LIN {X 0,Y 449.957,Z 720.436,A -85,B 0,C 180,E1 -8545.011,E2 -8545.011} C_VEL
LIN {X 0,Y 447.528,Z 720.738,A -85,B 0,C 180,E1 -8545.981,E2 -8545.981} C_VEL
LIN {X 0,Y 446.586,Z 720.854,A -85,B 0,C 180,E1 -8546.732,E2 -8546.732} C_VEL
LIN {X 0,Y 446.564,Z 720.858,A -85,B 0,C 180,E1 -8546.985,E2 -8546.985} C_VEL
LIN {X 0,Y 446.721,Z 720.839,A -85,B 0,C 180,E1 -8550,E2 -8550} C_VEL
LIN {X 0,Y 446.657,Z 720.845,A -85,B 0,C 180,E1 -8552.706,E2 -8552.706} C_VEL
LIN {X 0,Y 446.61,Z 720.852,A -85,B 0,C 180,E1 -8556.324,E2 -8556.324} C_VEL
LIN {X 0,Y 446.529,Z 720.861,A -85,B 0,C 180,E1 -8559.056,E2 -8559.056} C_VEL
LIN {X 0,Y 446.525,Z 720.861,A -85,B 0,C 180,E1 -8562.73,E2 -8562.73} C_VEL
LIN {X 0,Y 446.499,Z 720.866,A -85,B 0,C 180,E1 -8566.227,E2 -8566.227} C_VEL
LIN {X 0,Y 446.472,Z 720.868,A -85,B 0,C 180,E1 -8569.303,E2 -8569.303} C_VEL
LIN {X 0,Y 446.422,Z 720.877,A -85,B 0,C 180,E1 -8572.2,E2 -8572.2} C_VEL
LIN {X 0,Y 446.436,Z 720.872,A -85,B 0,C 180,E1 -8575.154,E2 -8575.154} C_VEL
LIN {X 0,Y 446.452,Z 720.875,A -85,B 0,C 180,E1 -8578.181,E2 -8578.181} C_VEL
LIN {X 0,Y 446.419,Z 720.873,A -85,B 0,C 180,E1 -8581.3,E2 -8581.3} C_VEL
LIN {X 0,Y 446.427,Z 720.876,A -85,B 0,C 180,E1 -8584.524,E2 -8584.524} C_VEL
LIN {X 0,Y 446.417,Z 720.878,A -85,B 0,C 180,E1 -8588.079,E2 -8588.079} C_VEL
LIN {X 0,Y 446.43,Z 720.873,A -85,B 0,C 180,E1 -8590.918,E2 -8590.918} C_VEL
LIN {X 0,Y 446.402,Z 720.876,A -85,B 0,C 180,E1 -8593.846,E2 -8593.846} C_VEL
LIN {X 0,Y 446.452,Z 720.961,A -85,B 0,C 180,E1 -8596.869,E2 -8596.869} C_VEL
LIN {X 0,Y 449.623,Z 732.094,A -85,B 0,C 180,E1 -8597.609,E2 -8597.609} C_VEL
LIN {X 0,Y 449.235,Z 743.341,A -85,B 0,C 180,E1 -8598.404,E2 -8598.404} C_VEL
LIN {X 0,Y 448.757,Z 753.702,A -85,B 0,C 180,E1 -8599.315,E2 -8599.315} C_VEL
LIN {X 0,Y 448.366,Z 763.491,A -85,B 0,C 180,E1 -8600.377,E2 -8600.377} C_VEL
LIN {X 0,Y 447.923,Z 771.722,A -85,B 0,C 180,E1 -8601.459,E2 -8601.459} C_VEL
LIN {X 0,Y 447.455,Z 779.986,A -85,B 0,C 180,E1 -8602.793,E2 -8602.793} C_VEL
LIN {X 0,Y 447.1,Z 786.808,A -85,B 0,C 180,E1 -8604.159,E2 -8604.159} C_VEL
LIN {X 0,Y 446.771,Z 792.209,A -85,B 0,C 180,E1 -8605.507,E2 -8605.507} C_VEL
LIN {X 0,Y 446.539,Z 797.152,A -85,B 0,C 180,E1 -8607.112,E2 -8607.112} C_VEL
LIN {X 0,Y 446.389,Z 800.563,A -85,B 0,C 180,E1 -8608.697,E2 -8608.697} C_VEL
LIN {X 0,Y 446.309,Z 802.432,A -85,B 0,C 180,E1 -8610.007,E2 -8610.007} C_VEL
LIN {X 0,Y 446.237,Z 803.608,A -85,B 0,C 180,E1 -8611.804,E2 -8611.804} C_VEL
LIN {X 0,Y 446.27,Z 803.599,A -85,B 0,C 180,E1 -8612.825,E2 -8612.825} C_VEL
LIN {X 0,Y 446.323,Z 803.053,A -85,B 0,C 180,E1 -8613.838,E2 -8613.838} C_VEL
LIN {X 0,Y 446.441,Z 802.052,A -85,B 0,C 180,E1 -8614.846,E2 -8614.846} C_VEL
LIN {X 0,Y 446.586,Z 800.438,A -85,B 0,C 180,E1 -8615.89,E2 -8615.89} C_VEL
LIN {X 0,Y 446.808,Z 797.298,A -85,B 0,C 180,E1 -8617.333,E2 -8617.333} C_VEL
LIN {X 0,Y 447.056,Z 792.895,A -85,B 0,C 180,E1 -8618.803,E2 -8618.803} C_VEL
LIN {X 0,Y 447.453,Z 787.514,A -85,B 0,C 180,E1 -8620.179,E2 -8620.179} C_VEL
LIN {X 0,Y 447.845,Z 781.194,A -85,B 0,C 180,E1 -8621.471,E2 -8621.471} C_VEL
LIN {X 0,Y 448.324,Z 773.951,A -85,B 0,C 180,E1 -8622.671,E2 -8622.671} C_VEL
LIN {X 0,Y 448.853,Z 765.107,A -85,B 0,C 180,E1 -8623.863,E2 -8623.863} C_VEL
LIN {X 0,Y 449.328,Z 755.427,A -85,B 0,C 180,E1 -8624.928,E2 -8624.928} C_VEL
LIN {X 0,Y 449.737,Z 745.469,A -85,B 0,C 180,E1 -8625.818,E2 -8625.818} C_VEL
LIN {X 0,Y 450.116,Z 734.981,A -85,B 0,C 180,E1 -8626.57,E2 -8626.57} C_VEL
LIN {X 0,Y 449.749,Z 731.701,A -85,B 0,C 180,E1 -8626.789,E2 -8626.789} C_VEL
LIN {X 0,Y 446.534,Z 720.868,A -85,B 0,C 180,E1 -8627.52,E2 -8627.52} C_VEL
LIN {X 0,Y 446.537,Z 720.862,A -85,B 0,C 180,E1 -8630.944,E2 -8630.944} C_VEL
LIN {X 0,Y 446.617,Z 720.854,A -85,B 0,C 180,E1 -8633.676,E2 -8633.676} C_VEL
LIN {X 0,Y 446.686,Z 720.845,A -85,B 0,C 180,E1 -8637.294,E2 -8637.294} C_VEL
LIN {X 0,Y 446.794,Z 720.832,A -85,B 0,C 180,E1 -8640,E2 -8640} C_VEL
LIN {X 0,Y 446.687,Z 720.837,A -85,B 0,C 180,E1 -8642.705,E2 -8642.705} C_VEL
LIN {X 0,Y 446.641,Z 720.849,A -85,B 0,C 180,E1 -8646.324,E2 -8646.324} C_VEL
LIN {X 0,Y 446.536,Z 720.854,A -85,B 0,C 180,E1 -8649.055,E2 -8649.055} C_VEL
LIN {X 0,Y 446.525,Z 720.861,A -85,B 0,C 180,E1 -8652.73,E2 -8652.73} C_VEL
LIN {X 0,Y 446.5,Z 720.87,A -85,B 0,C 180,E1 -8656.228,E2 -8656.228} C_VEL
LIN {X 0,Y 446.472,Z 720.867,A -85,B 0,C 180,E1 -8659.303,E2 -8659.303} C_VEL
LIN {X 0,Y 446.422,Z 720.878,A -85,B 0,C 180,E1 -8662.199,E2 -8662.199} C_VEL
LIN {X 0,Y 446.448,Z 720.871,A -85,B 0,C 180,E1 -8665.153,E2 -8665.153} C_VEL
LIN {X 0,Y 446.488,Z 720.871,A -85,B 0,C 180,E1 -8668.178,E2 -8668.178} C_VEL
LIN {X 0,Y 446.423,Z 720.874,A -85,B 0,C 180,E1 -8671.775,E2 -8671.775} C_VEL
LIN {X 0,Y 446.433,Z 720.878,A -85,B 0,C 180,E1 -8674.523,E2 -8674.523} C_VEL
LIN {X 0,Y 446.419,Z 720.88,A -85,B 0,C 180,E1 -8678.079,E2 -8678.079} C_VEL
LIN {X 0,Y 446.43,Z 720.881,A -85,B 0,C 180,E1 -8680.917,E2 -8680.917} C_VEL
LIN {X 0,Y 446.405,Z 720.88,A -85,B 0,C 180,E1 -8683.846,E2 -8683.846} C_VEL
LIN {X 0,Y 446.403,Z 720.882,A -85,B 0,C 180,E1 -8686.403,E2 -8686.403} C_VEL
LIN {X 0,Y 446.446,Z 720.918,A -85,B 0,C 180,E1 -8688.46,E2 -8688.46} C_VEL
LIN {X 0,Y 448.073,Z 729.07,A -85,B 0,C 180,E1 -8691.141,E2 -8691.141} C_VEL
LIN {X 0,Y 449.284,Z 735.97,A -85,B 0,C 180,E1 -8693.241,E2 -8693.241} C_VEL
LIN {X 0,Y 448.846,Z 744.926,A -85,B 0,C 180,E1 -8695.689,E2 -8695.689} C_VEL
LIN {X 0,Y 448.24,Z 757.053,A -85,B 0,C 180,E1 -8698.841,E2 -8698.841} C_VEL
LIN {X 0,Y 447.623,Z 771.408,A -85,B 0,C 180,E1 -8702.408,E2 -8702.408} C_VEL
LIN {X 0,Y 447.2,Z 783.707,A -85,B 0,C 180,E1 -8705.358,E2 -8705.358} C_VEL
LIN {X 0,Y 446.783,Z 798.343,A -85,B 0,C 180,E1 -8708.789,E2 -8708.789} C_VEL
LIN {X 0,Y 446.408,Z 813.869,A -85,B 0,C 180,E1 -8712.358,E2 -8712.358} C_VEL
LIN {X 0,Y 446.248,Z 820.18,A -85,B 0,C 180,E1 -8713.796,E2 -8713.796} C_VEL
LIN {X 0,Y 447.563,Z 835.272,A -85,B 0,C 180,E1 -8714.244,E2 -8714.244} C_VEL
LIN {X 0,Y 448.738,Z 846.604,A -85,B 0,C 180,E1 -8714.733,E2 -8714.733} C_VEL
LIN {X 0,Y 448.868,Z 851.343,A -85,B 0,C 180,E1 -8714.97,E2 -8714.97} C_VEL
LIN {X 0,Y 448.236,Z 863.895,A -85,B 0,C 180,E1 -8715.703,E2 -8715.703} C_VEL
LIN {X 0,Y 447.652,Z 875.363,A -85,B 0,C 180,E1 -8716.572,E2 -8716.572} C_VEL
LIN {X 0,Y 447.242,Z 885.483,A -85,B 0,C 180,E1 -8717.522,E2 -8717.522} C_VEL
LIN {X 0,Y 446.788,Z 893.591,A -85,B 0,C 180,E1 -8718.43,E2 -8718.43} C_VEL
LIN {X 0,Y 446.292,Z 903.634,A -85,B 0,C 180,E1 -8719.795,E2 -8719.795} C_VEL
LIN {X 0,Y 446.004,Z 911.698,A -85,B 0,C 180,E1 -8721.162,E2 -8721.162} C_VEL
LIN {X 0,Y 445.853,Z 917.231,A -85,B 0,C 180,E1 -8722.3,E2 -8722.3} C_VEL
LIN {X 0,Y 445.791,Z 922.628,A -85,B 0,C 180,E1 -8723.664,E2 -8723.664} C_VEL
LIN {X 0,Y 445.738,Z 926.828,A -85,B 0,C 180,E1 -8725.025,E2 -8725.025} C_VEL
LIN {X 0,Y 445.732,Z 929.95,A -85,B 0,C 180,E1 -8726.384,E2 -8726.384} C_VEL
LIN {X 0,Y 445.696,Z 931.439,A -85,B 0,C 180,E1 -8727.288,E2 -8727.288} C_VEL
LIN {X 0,Y 445.69,Z 932.518,A -85,B 0,C 180,E1 -8728.193,E2 -8728.193} C_VEL
LIN {X 0,Y 445.662,Z 933.188,A -85,B 0,C 180,E1 -8729.096,E2 -8729.096} C_VEL
LIN {X 0,Y 445.653,Z 933.446,A -85,B 0,C 180,E1 -8730,E2 -8730} C_VEL
LIN {X 0,Y 445.653,Z 933.252,A -85,B 0,C 180,E1 -8730.904,E2 -8730.904} C_VEL
LIN {X 0,Y 445.673,Z 932.66,A -85,B 0,C 180,E1 -8731.807,E2 -8731.807} C_VEL
LIN {X 0,Y 445.675,Z 931.66,A -85,B 0,C 180,E1 -8732.711,E2 -8732.711} C_VEL
LIN {X 0,Y 445.73,Z 930.242,A -85,B 0,C 180,E1 -8733.616,E2 -8733.616} C_VEL
LIN {X 0,Y 445.693,Z 927.234,A -85,B 0,C 180,E1 -8734.975,E2 -8734.975} C_VEL
LIN {X 0,Y 445.708,Z 922.253,A -85,B 0,C 180,E1 -8736.588,E2 -8736.588} C_VEL
LIN {X 0,Y 445.895,Z 915.848,A -85,B 0,C 180,E1 -8738.155,E2 -8738.155} C_VEL
LIN {X 0,Y 446.119,Z 908.774,A -85,B 0,C 180,E1 -8739.521,E2 -8739.521} C_VEL
LIN {X 0,Y 446.523,Z 899.934,A -85,B 0,C 180,E1 -8740.887,E2 -8740.887} C_VEL
LIN {X 0,Y 446.967,Z 890.906,A -85,B 0,C 180,E1 -8742.025,E2 -8742.025} C_VEL
LIN {X 0,Y 447.505,Z 881.147,A -85,B 0,C 180,E1 -8743.035,E2 -8743.035} C_VEL
LIN {X 0,Y 448.02,Z 870.196,A -85,B 0,C 180,E1 -8743.956,E2 -8743.956} C_VEL
LIN {X 0,Y 448.715,Z 858.163,A -85,B 0,C 180,E1 -8744.745,E2 -8744.745} C_VEL
LIN {X 0,Y 449.042,Z 848.273,A -85,B 0,C 180,E1 -8745.256,E2 -8745.256} C_VEL
LIN {X 0,Y 447.601,Z 835.432,A -85,B 0,C 180,E1 -8745.801,E2 -8745.801} C_VEL
LIN {X 0,Y 446.271,Z 822.393,A -85,B 0,C 180,E1 -8746.2,E2 -8746.2} C_VEL
LIN {X 0,Y 446.563,Z 811.414,A -85,B 0,C 180,E1 -8748.789,E2 -8748.789} C_VEL
LIN {X 0,Y 447.056,Z 797.262,A -85,B 0,C 180,E1 -8752.166,E2 -8752.166} C_VEL
LIN {X 0,Y 447.537,Z 785.194,A -85,B 0,C 180,E1 -8755.087,E2 -8755.087} C_VEL
LIN {X 0,Y 448.116,Z 773.165,A -85,B 0,C 180,E1 -8758.067,E2 -8758.067} C_VEL
LIN {X 0,Y 448.82,Z 760.067,A -85,B 0,C 180,E1 -8761.376,E2 -8761.376} C_VEL
LIN {X 0,Y 449.597,Z 748.02,A -85,B 0,C 180,E1 -8764.517,E2 -8764.517} C_VEL
LIN {X 0,Y 450.055,Z 739.541,A -85,B 0,C 180,E1 -8766.789,E2 -8766.789} C_VEL
LIN {X 0,Y 448.864,Z 732.725,A -85,B 0,C 180,E1 -8768.777,E2 -8768.777} C_VEL
LIN {X 0,Y 446.947,Z 723.206,A -85,B 0,C 180,E1 -8771.676,E2 -8771.676} C_VEL
LIN {X 0,Y 446.47,Z 720.873,A -85,B 0,C 180,E1 -8772.453,E2 -8772.453} C_VEL
LIN {X 0,Y 446.455,Z 720.874,A -85,B 0,C 180,E1 -8775.103,E2 -8775.103} C_VEL
LIN {X 0,Y 446.43,Z 720.874,A -85,B 0,C 180,E1 -8778.609,E2 -8778.609} C_VEL
LIN {X 0,Y 446.446,Z 720.873,A -85,B 0,C 180,E1 -8780.973,E2 -8780.973} C_VEL
LIN {X 0,Y 446.421,Z 720.873,A -85,B 0,C 180,E1 -8784.374,E2 -8784.374} C_VEL
LIN {X 0,Y 446.424,Z 720.88,A -85,B 0,C 180,E1 -8787.639,E2 -8787.639} C_VEL
LIN {X 0,Y 446.451,Z 720.87,A -85,B 0,C 180,E1 -8790.791,E2 -8790.791} C_VEL
LIN {X 0,Y 446.48,Z 720.872,A -85,B 0,C 180,E1 -8793.849,E2 -8793.849} C_VEL
LIN {X 0,Y 446.429,Z 720.873,A -85,B 0,C 180,E1 -8796.823,E2 -8796.823} C_VEL
LIN {X 0,Y 446.446,Z 720.875,A -85,B 0,C 180,E1 -8799.737,E2 -8799.737} C_VEL
LIN {X 0,Y 446.46,Z 720.87,A -85,B 0,C 180,E1 -8802.597,E2 -8802.597} C_VEL
LIN {X 0,Y 446.473,Z 720.869,A -85,B 0,C 180,E1 -8805.413,E2 -8805.413} C_VEL
LIN {X 0,Y 446.52,Z 720.867,A -85,B 0,C 180,E1 -8808.193,E2 -8808.193} C_VEL
LIN {X 0,Y 446.603,Z 720.854,A -85,B 0,C 180,E1 -8811.858,E2 -8811.858} C_VEL
LIN {X 0,Y 446.645,Z 720.848,A -85,B 0,C 180,E1 -8814.583,E2 -8814.583} C_VEL
LIN {X 0,Y 446.663,Z 720.848,A -85,B 0,C 180,E1 -8818.197,E2 -8818.197} C_VEL
LIN {X 0,Y 446.792,Z 720.831,A -85,B 0,C 180,E1 -8820,E2 -8820} C_VEL
LIN {X 0,Y 446.684,Z 720.844,A -85,B 0,C 180,E1 -8822.706,E2 -8822.706} C_VEL
LIN {X 0,Y 446.619,Z 720.853,A -85,B 0,C 180,E1 -8826.324,E2 -8826.324} C_VEL
LIN {X 0,Y 446.535,Z 720.861,A -85,B 0,C 180,E1 -8829.056,E2 -8829.056} C_VEL
LIN {X 0,Y 446.524,Z 720.866,A -85,B 0,C 180,E1 -8832.73,E2 -8832.73} C_VEL
LIN {X 0,Y 446.491,Z 720.869,A -85,B 0,C 180,E1 -8836.459,E2 -8836.459} C_VEL
LIN {X 0,Y 446.471,Z 720.869,A -85,B 0,C 180,E1 -8839.303,E2 -8839.303} C_VEL
LIN {X 0,Y 446.42,Z 720.877,A -85,B 0,C 180,E1 -8842.2,E2 -8842.2} C_VEL
LIN {X 0,Y 446.421,Z 720.877,A -85,B 0,C 180,E1 -8845.155,E2 -8845.155} C_VEL
LIN {X 0,Y 446.442,Z 720.875,A -85,B 0,C 180,E1 -8848.182,E2 -8848.182} C_VEL
LIN {X 0,Y 446.416,Z 720.877,A -85,B 0,C 180,E1 -8851.301,E2 -8851.301} C_VEL
LIN {X 0,Y 446.423,Z 720.877,A -85,B 0,C 180,E1 -8854.524,E2 -8854.524} C_VEL
LIN {X 0,Y 446.405,Z 720.878,A -85,B 0,C 180,E1 -8858.077,E2 -8858.077} C_VEL
LIN {X 0,Y 446.402,Z 720.88,A -85,B 0,C 180,E1 -8861.394,E2 -8861.394} C_VEL
LIN {X 0,Y 446.423,Z 720.877,A -85,B 0,C 180,E1 -8865.108,E2 -8865.108} C_VEL
LIN {X 0,Y 446.402,Z 720.881,A -85,B 0,C 180,E1 -8868.606,E2 -8868.606} C_VEL
LIN {X 0,Y 446.399,Z 720.878,A -85,B 0,C 180,E1 -8871.924,E2 -8871.924} C_VEL
LIN {X 0,Y 446.416,Z 720.878,A -85,B 0,C 180,E1 -8875.476,E2 -8875.476} C_VEL
LIN {X 0,Y 446.392,Z 720.882,A -85,B 0,C 180,E1 -8878.698,E2 -8878.698} C_VEL
LIN {X 0,Y 446.407,Z 720.878,A -85,B 0,C 180,E1 -8881.841,E2 -8881.841} C_VEL
LIN {X 0,Y 446.414,Z 720.879,A -85,B 0,C 180,E1 -8884.845,E2 -8884.845} C_VEL
LIN {X 0,Y 446.451,Z 720.872,A -85,B 0,C 180,E1 -8888.245,E2 -8888.245} C_VEL
LIN {X 0,Y 446.45,Z 720.873,A -85,B 0,C 180,E1 -8891.649,E2 -8891.649} C_VEL
LIN {X 0,Y 446.496,Z 720.866,A -85,B 0,C 180,E1 -8894.479,E2 -8894.479} C_VEL
LIN {X 0,Y 446.508,Z 720.865,A -85,B 0,C 180,E1 -8898.193,E2 -8898.193} C_VEL
LIN {X 0,Y 446.508,Z 720.866,A -85,B 0,C 180,E1 -8900.944,E2 -8900.944} C_VEL
LIN {X 0,Y 446.608,Z 720.854,A -85,B 0,C 180,E1 -8903.676,E2 -8903.676} C_VEL
LIN {X 0,Y 446.564,Z 720.858,A -85,B 0,C 180,E1 -8906.985,E2 -8906.985} C_VEL
LIN {X 0,Y 446.35,Z 720.888,A -85,B 0,C 180,E1 -8907.489,E2 -8907.489} C_VEL
LIN {X 0,Y 445.047,Z 721.052,A -85,B 0,C 180,E1 -8908.232,E2 -8908.232} C_VEL
LIN {X 0,Y 440.623,Z 721.602,A -85,B 0,C 180,E1 -8909.947,E2 -8909.947} C_VEL
LIN {X 0,Y 439.571,Z 721.729,A -85,B 0,C 180,E1 -8910.711,E2 -8910.711} C_VEL
LIN {X 0,Y 439.505,Z 721.736,A -85,B 0,C 180,E1 -8910.97,E2 -8910.97} C_VEL
LIN {X 0,Y 439.609,Z 721.723,A -85,B 0,C 180,E1 -8912.749,E2 -8912.749} C_VEL
LIN {X 0,Y 439.563,Z 721.73,A -85,B 0,C 180,E1 -8916.426,E2 -8916.426} C_VEL
LIN {X 0,Y 439.494,Z 721.738,A -85,B 0,C 180,E1 -8919.202,E2 -8919.202} C_VEL
LIN {X 0,Y 439.469,Z 721.74,A -85,B 0,C 180,E1 -8922.938,E2 -8922.938} C_VEL
LIN {X 0,Y 439.45,Z 721.744,A -85,B 0,C 180,E1 -8926.348,E2 -8926.348} C_VEL
LIN {X 0,Y 439.406,Z 721.751,A -85,B 0,C 180,E1 -8929.626,E2 -8929.626} C_VEL
LIN {X 0,Y 439.367,Z 721.753,A -85,B 0,C 180,E1 -8932.576,E2 -8932.576} C_VEL
LIN {X 0,Y 439.376,Z 721.753,A -85,B 0,C 180,E1 -8935.587,E2 -8935.587} C_VEL
LIN {X 0,Y 439.403,Z 721.749,A -85,B 0,C 180,E1 -8938.675,E2 -8938.675} C_VEL
LIN {X 0,Y 439.372,Z 721.756,A -85,B 0,C 180,E1 -8942.03,E2 -8942.03} C_VEL
LIN {X 0,Y 439.396,Z 721.748,A -85,B 0,C 180,E1 -8945.34,E2 -8945.34} C_VEL
LIN {X 0,Y 439.379,Z 721.754,A -85,B 0,C 180,E1 -8948.596,E2 -8948.596} C_VEL
LIN {X 0,Y 439.392,Z 721.748,A -85,B 0,C 180,E1 -8951.257,E2 -8951.257} C_VEL
LIN {X 0,Y 439.403,Z 721.752,A -85,B 0,C 180,E1 -8954.729,E2 -8954.729} C_VEL
LIN {X 0,Y 439.378,Z 721.763,A -85,B 0,C 180,E1 -8956.638,E2 -8956.638} C_VEL
LIN {X 0,Y 442.712,Z 733.524,A -85,B 0,C 180,E1 -8957.437,E2 -8957.437} C_VEL
LIN {X 0,Y 442.343,Z 745.457,A -85,B 0,C 180,E1 -8958.309,E2 -8958.309} C_VEL
LIN {X 0,Y 441.848,Z 756.239,A -85,B 0,C 180,E1 -8959.296,E2 -8959.296} C_VEL
LIN {X 0,Y 441.356,Z 766.209,A -85,B 0,C 180,E1 -8960.435,E2 -8960.435} C_VEL
LIN {X 0,Y 440.908,Z 774.318,A -85,B 0,C 180,E1 -8961.563,E2 -8961.563} C_VEL
LIN {X 0,Y 440.402,Z 782.389,A -85,B 0,C 180,E1 -8962.931,E2 -8962.931} C_VEL
LIN {X 0,Y 440.084,Z 788.71,A -85,B 0,C 180,E1 -8964.261,E2 -8964.261} C_VEL
LIN {X 0,Y 439.777,Z 793.254,A -85,B 0,C 180,E1 -8965.436,E2 -8965.436} C_VEL
LIN {X 0,Y 439.539,Z 798.2,A -85,B 0,C 180,E1 -8967.068,E2 -8967.068} C_VEL
LIN {X 0,Y 439.45,Z 800.616,A -85,B 0,C 180,E1 -8968.146,E2 -8968.146} C_VEL
LIN {X 0,Y 439.302,Z 803.199,A -85,B 0,C 180,E1 -8969.758,E2 -8969.758} C_VEL
LIN {X 0,Y 439.213,Z 804.607,A -85,B 0,C 180,E1 -8971.652,E2 -8971.652} C_VEL
LIN {X 0,Y 439.283,Z 804.438,A -85,B 0,C 180,E1 -8973.386,E2 -8973.386} C_VEL
LIN {X 0,Y 439.387,Z 803.656,A -85,B 0,C 180,E1 -8974.414,E2 -8974.414} C_VEL
LIN {X 0,Y 439.555,Z 801.993,A -85,B 0,C 180,E1 -8975.696,E2 -8975.696} C_VEL
LIN {X 0,Y 439.732,Z 799.551,A -85,B 0,C 180,E1 -8976.948,E2 -8976.948} C_VEL
LIN {X 0,Y 440.019,Z 795.551,A -85,B 0,C 180,E1 -8978.447,E2 -8978.447} C_VEL
LIN {X 0,Y 440.394,Z 790.266,A -85,B 0,C 180,E1 -8979.924,E2 -8979.924} C_VEL
LIN {X 0,Y 440.878,Z 783.437,A -85,B 0,C 180,E1 -8981.408,E2 -8981.408} C_VEL
LIN {X 0,Y 441.45,Z 775.445,A -85,B 0,C 180,E1 -8982.789,E2 -8982.789} C_VEL
LIN {X 0,Y 442.028,Z 766.039,A -85,B 0,C 180,E1 -8984.082,E2 -8984.082} C_VEL
LIN {X 0,Y 442.545,Z 756.341,A -85,B 0,C 180,E1 -8985.162,E2 -8985.162} C_VEL
LIN {X 0,Y 442.99,Z 746.057,A -85,B 0,C 180,E1 -8986.092,E2 -8986.092} C_VEL
LIN {X 0,Y 443.294,Z 734.557,A -85,B 0,C 180,E1 -8986.914,E2 -8986.914} C_VEL
LIN {X 0,Y 439.771,Z 723.032,A -85,B 0,C 180,E1 -8987.726,E2 -8987.726} C_VEL
LIN {X 0,Y 439.473,Z 721.747,A -85,B 0,C 180,E1 -8987.824,E2 -8987.824} C_VEL
LIN {X 0,Y 439.5,Z 721.738,A -85,B 0,C 180,E1 -8990.798,E2 -8990.798} C_VEL
LIN {X 0,Y 439.59,Z 721.731,A -85,B 0,C 180,E1 -8993.574,E2 -8993.574} C_VEL
LIN {X 0,Y 439.636,Z 721.723,A -85,B 0,C 180,E1 -8997.251,E2 -8997.251} C_VEL
LIN {X 0,Y 439.763,Z 721.708,A -85,B 0,C 180,E1 -9000,E2 -9000} C_VEL
LIN {X 0,Y 439.636,Z 721.715,A -85,B 0,C 180,E1 -9002.749,E2 -9002.749} C_VEL
LIN {X 0,Y 439.613,Z 721.723,A -85,B 0,C 180,E1 -9006.425,E2 -9006.425} C_VEL
LIN {X 0,Y 439.499,Z 721.731,A -85,B 0,C 180,E1 -9009.202,E2 -9009.202} C_VEL
LIN {X 0,Y 439.469,Z 721.739,A -85,B 0,C 180,E1 -9012.937,E2 -9012.937} C_VEL
LIN {X 0,Y 439.45,Z 721.747,A -85,B 0,C 180,E1 -9016.348,E2 -9016.348} C_VEL
LIN {X 0,Y 439.406,Z 721.749,A -85,B 0,C 180,E1 -9019.626,E2 -9019.626} C_VEL
LIN {X 0,Y 439.368,Z 721.755,A -85,B 0,C 180,E1 -9022.575,E2 -9022.575} C_VEL
LIN {X 0,Y 439.401,Z 721.749,A -85,B 0,C 180,E1 -9025.585,E2 -9025.585} C_VEL
LIN {X 0,Y 439.421,Z 721.747,A -85,B 0,C 180,E1 -9028.673,E2 -9028.673} C_VEL
LIN {X 0,Y 439.374,Z 721.754,A -85,B 0,C 180,E1 -9032.03,E2 -9032.03} C_VEL
LIN {X 0,Y 439.398,Z 721.751,A -85,B 0,C 180,E1 -9035.34,E2 -9035.34} C_VEL
LIN {X 0,Y 439.386,Z 721.757,A -85,B 0,C 180,E1 -9038.595,E2 -9038.595} C_VEL
LIN {X 0,Y 439.391,Z 721.755,A -85,B 0,C 180,E1 -9041.257,E2 -9041.257} C_VEL
LIN {X 0,Y 439.404,Z 721.753,A -85,B 0,C 180,E1 -9044.729,E2 -9044.729} C_VEL
LIN {X 0,Y 439.411,Z 721.835,A -85,B 0,C 180,E1 -9048.097,E2 -9048.097} C_VEL
LIN {X 0,Y 441.078,Z 730.102,A -85,B 0,C 180,E1 -9050.898,E2 -9050.898} C_VEL
LIN {X 0,Y 442.2,Z 736.316,A -85,B 0,C 180,E1 -9052.847,E2 -9052.847} C_VEL
LIN {X 0,Y 442.225,Z 740.828,A -85,B 0,C 180,E1 -9054.146,E2 -9054.146} C_VEL
LIN {X 0,Y 441.498,Z 753.283,A -85,B 0,C 180,E1 -9057.531,E2 -9057.531} C_VEL
LIN {X 0,Y 440.814,Z 766.292,A -85,B 0,C 180,E1 -9060.883,E2 -9060.883} C_VEL
LIN {X 0,Y 440.313,Z 779.726,A -85,B 0,C 180,E1 -9064.218,E2 -9064.218} C_VEL
LIN {X 0,Y 439.843,Z 793.157,A -85,B 0,C 180,E1 -9067.45,E2 -9067.45} C_VEL
LIN {X 0,Y 439.447,Z 805.532,A -85,B 0,C 180,E1 -9070.376,E2 -9070.376} C_VEL
LIN {X 0,Y 439.227,Z 816.87,A -85,B 0,C 180,E1 -9073.021,E2 -9073.021} C_VEL
LIN {X 0,Y 439.185,Z 818.992,A -85,B 0,C 180,E1 -9073.513,E2 -9073.513} C_VEL
LIN {X 0,Y 440.509,Z 833.536,A -85,B 0,C 180,E1 -9073.957,E2 -9073.957} C_VEL
LIN {X 0,Y 441.424,Z 844.174,A -85,B 0,C 180,E1 -9074.415,E2 -9074.415} C_VEL
LIN {X 0,Y 441.96,Z 850.208,A -85,B 0,C 180,E1 -9074.729,E2 -9074.729} C_VEL
LIN {X 0,Y 441.302,Z 862.746,A -85,B 0,C 180,E1 -9075.473,E2 -9075.473} C_VEL
LIN {X 0,Y 440.656,Z 874.622,A -85,B 0,C 180,E1 -9076.391,E2 -9076.391} C_VEL
LIN {X 0,Y 440.214,Z 884.341,A -85,B 0,C 180,E1 -9077.319,E2 -9077.319} C_VEL
LIN {X 0,Y 439.684,Z 894.309,A -85,B 0,C 180,E1 -9078.474,E2 -9078.474} C_VEL
LIN {X 0,Y 439.248,Z 902.523,A -85,B 0,C 180,E1 -9079.63,E2 -9079.63} C_VEL
LIN {X 0,Y 438.943,Z 910.604,A -85,B 0,C 180,E1 -9081.019,E2 -9081.019} C_VEL
LIN {X 0,Y 438.797,Z 916.153,A -85,B 0,C 180,E1 -9082.175,E2 -9082.175} C_VEL
LIN {X 0,Y 438.711,Z 921.56,A -85,B 0,C 180,E1 -9083.561,E2 -9083.561} C_VEL
LIN {X 0,Y 438.699,Z 925.78,A -85,B 0,C 180,E1 -9084.945,E2 -9084.945} C_VEL
LIN {X 0,Y 438.696,Z 928.914,A -85,B 0,C 180,E1 -9086.326,E2 -9086.326} C_VEL
LIN {X 0,Y 438.657,Z 930.412,A -85,B 0,C 180,E1 -9087.245,E2 -9087.245} C_VEL
LIN {X 0,Y 438.656,Z 931.498,A -85,B 0,C 180,E1 -9088.164,E2 -9088.164} C_VEL
LIN {X 0,Y 438.632,Z 932.174,A -85,B 0,C 180,E1 -9089.082,E2 -9089.082} C_VEL
LIN {X 0,Y 438.625,Z 932.438,A -85,B 0,C 180,E1 -9090,E2 -9090} C_VEL
LIN {X 0,Y 438.622,Z 932.251,A -85,B 0,C 180,E1 -9090.918,E2 -9090.918} C_VEL
LIN {X 0,Y 438.636,Z 931.661,A -85,B 0,C 180,E1 -9091.836,E2 -9091.836} C_VEL
LIN {X 0,Y 438.635,Z 930.663,A -85,B 0,C 180,E1 -9092.755,E2 -9092.755} C_VEL
LIN {X 0,Y 438.694,Z 929.246,A -85,B 0,C 180,E1 -9093.674,E2 -9093.674} C_VEL
LIN {X 0,Y 438.637,Z 926.236,A -85,B 0,C 180,E1 -9095.056,E2 -9095.056} C_VEL
LIN {X 0,Y 438.645,Z 921.585,A -85,B 0,C 180,E1 -9096.6,E2 -9096.6} C_VEL
LIN {X 0,Y 438.795,Z 915.864,A -85,B 0,C 180,E1 -9098.056,E2 -9098.056} C_VEL
LIN {X 0,Y 439.017,Z 909.013,A -85,B 0,C 180,E1 -9099.444,E2 -9099.444} C_VEL
LIN {X 0,Y 439.393,Z 900.532,A -85,B 0,C 180,E1 -9100.832,E2 -9100.832} C_VEL
LIN {X 0,Y 439.834,Z 891.819,A -85,B 0,C 180,E1 -9101.989,E2 -9101.989} C_VEL
LIN {X 0,Y 440.377,Z 882.425,A -85,B 0,C 180,E1 -9103.017,E2 -9103.017} C_VEL
LIN {X 0,Y 440.993,Z 870.583,A -85,B 0,C 180,E1 -9104.066,E2 -9104.066} C_VEL
LIN {X 0,Y 441.7,Z 859.025,A -85,B 0,C 180,E1 -9104.867,E2 -9104.867} C_VEL
LIN {X 0,Y 441.97,Z 848.392,A -85,B 0,C 180,E1 -9105.447,E2 -9105.447} C_VEL
LIN {X 0,Y 440.612,Z 835.394,A -85,B 0,C 180,E1 -9106.019,E2 -9106.019} C_VEL
LIN {X 0,Y 439.2,Z 821.487,A -85,B 0,C 180,E1 -9106.466,E2 -9106.466} C_VEL
LIN {X 0,Y 439.501,Z 810.893,A -85,B 0,C 180,E1 -9109.012,E2 -9109.012} C_VEL
LIN {X 0,Y 439.985,Z 798.138,A -85,B 0,C 180,E1 -9112.112,E2 -9112.112} C_VEL
LIN {X 0,Y 440.597,Z 784.405,A -85,B 0,C 180,E1 -9115.511,E2 -9115.511} C_VEL
LIN {X 0,Y 441.178,Z 772.372,A -85,B 0,C 180,E1 -9118.549,E2 -9118.549} C_VEL
LIN {X 0,Y 441.879,Z 760.325,A -85,B 0,C 180,E1 -9121.659,E2 -9121.659} C_VEL
LIN {X 0,Y 442.724,Z 748.25,A -85,B 0,C 180,E1 -9124.854,E2 -9124.854} C_VEL
LIN {X 0,Y 443.078,Z 740.212,A -85,B 0,C 180,E1 -9127.067,E2 -9127.067} C_VEL
LIN {X 0,Y 441.442,Z 731.865,A -85,B 0,C 180,E1 -9129.555,E2 -9129.555} C_VEL
LIN {X 0,Y 439.404,Z 721.753,A -85,B 0,C 180,E1 -9132.78,E2 -9132.78} C_VEL
LIN {X 0,Y 439.369,Z 721.754,A -85,B 0,C 180,E1 -9136.039,E2 -9136.039} C_VEL
LIN {X 0,Y 439.382,Z 721.755,A -85,B 0,C 180,E1 -9139.019,E2 -9139.019} C_VEL
LIN {X 0,Y 439.376,Z 721.757,A -85,B 0,C 180,E1 -9141.608,E2 -9141.608} C_VEL
LIN {X 0,Y 439.401,Z 721.748,A -85,B 0,C 180,E1 -9144.844,E2 -9144.844} C_VEL
LIN {X 0,Y 439.375,Z 721.753,A -85,B 0,C 180,E1 -9148.14,E2 -9148.14} C_VEL
LIN {X 0,Y 439.434,Z 721.749,A -85,B 0,C 180,E1 -9151.598,E2 -9151.598} C_VEL
LIN {X 0,Y 439.399,Z 721.749,A -85,B 0,C 180,E1 -9154.415,E2 -9154.415} C_VEL
LIN {X 0,Y 439.366,Z 721.754,A -85,B 0,C 180,E1 -9157.425,E2 -9157.425} C_VEL
LIN {X 0,Y 439.443,Z 721.743,A -85,B 0,C 180,E1 -9160.663,E2 -9160.663} C_VEL
LIN {X 0,Y 439.465,Z 721.744,A -85,B 0,C 180,E1 -9164.225,E2 -9164.225} C_VEL
LIN {X 0,Y 439.486,Z 721.743,A -85,B 0,C 180,E1 -9168.001,E2 -9168.001} C_VEL
LIN {X 0,Y 439.55,Z 721.732,A -85,B 0,C 180,E1 -9171.726,E2 -9171.726} C_VEL
LIN {X 0,Y 439.62,Z 721.724,A -85,B 0,C 180,E1 -9174.496,E2 -9174.496} C_VEL
LIN {X 0,Y 439.633,Z 721.724,A -85,B 0,C 180,E1 -9178.168,E2 -9178.168} C_VEL
LIN {X 0,Y 439.761,Z 721.706,A -85,B 0,C 180,E1 -9180,E2 -9180} C_VEL
LIN {X 0,Y 439.634,Z 721.722,A -85,B 0,C 180,E1 -9182.749,E2 -9182.749} C_VEL
LIN {X 0,Y 439.591,Z 721.73,A -85,B 0,C 180,E1 -9186.426,E2 -9186.426} C_VEL
LIN {X 0,Y 439.498,Z 721.738,A -85,B 0,C 180,E1 -9189.202,E2 -9189.202} C_VEL
LIN {X 0,Y 439.468,Z 721.743,A -85,B 0,C 180,E1 -9192.938,E2 -9192.938} C_VEL
LIN {X 0,Y 439.449,Z 721.745,A -85,B 0,C 180,E1 -9196.348,E2 -9196.348} C_VEL
LIN {X 0,Y 439.404,Z 721.75,A -85,B 0,C 180,E1 -9199.626,E2 -9199.626} C_VEL
LIN {X 0,Y 439.365,Z 721.756,A -85,B 0,C 180,E1 -9202.576,E2 -9202.576} C_VEL
LIN {X 0,Y 439.367,Z 721.754,A -85,B 0,C 180,E1 -9205.587,E2 -9205.587} C_VEL
LIN {X 0,Y 439.398,Z 721.752,A -85,B 0,C 180,E1 -9208.675,E2 -9208.675} C_VEL
LIN {X 0,Y 439.368,Z 721.755,A -85,B 0,C 180,E1 -9212.03,E2 -9212.03} C_VEL
LIN {X 0,Y 439.392,Z 721.753,A -85,B 0,C 180,E1 -9215.34,E2 -9215.34} C_VEL
LIN {X 0,Y 439.358,Z 721.757,A -85,B 0,C 180,E1 -9218.598,E2 -9218.598} C_VEL
LIN {X 0,Y 439.35,Z 721.758,A -85,B 0,C 180,E1 -9222.21,E2 -9222.21} C_VEL
LIN {X 0,Y 439.377,Z 721.755,A -85,B 0,C 180,E1 -9225.267,E2 -9225.267} C_VEL
LIN {X 0,Y 439.364,Z 721.756,A -85,B 0,C 180,E1 -9228.747,E2 -9228.747} C_VEL
LIN {X 0,Y 439.358,Z 721.757,A -85,B 0,C 180,E1 -9231.611,E2 -9231.611} C_VEL
LIN {X 0,Y 439.391,Z 721.753,A -85,B 0,C 180,E1 -9234.843,E2 -9234.843} C_VEL
LIN {X 0,Y 439.347,Z 721.757,A -85,B 0,C 180,E1 -9238.137,E2 -9238.137} C_VEL
LIN {X 0,Y 439.382,Z 721.753,A -85,B 0,C 180,E1 -9241.324,E2 -9241.324} C_VEL
LIN {X 0,Y 439.355,Z 721.756,A -85,B 0,C 180,E1 -9244.412,E2 -9244.412} C_VEL
LIN {X 0,Y 439.365,Z 721.755,A -85,B 0,C 180,E1 -9247.425,E2 -9247.425} C_VEL
LIN {X 0,Y 439.444,Z 721.745,A -85,B 0,C 180,E1 -9250.663,E2 -9250.663} C_VEL
LIN {X 0,Y 439.457,Z 721.743,A -85,B 0,C 180,E1 -9254.224,E2 -9254.224} C_VEL
LIN {X 0,Y 439.478,Z 721.741,A -85,B 0,C 180,E1 -9258.001,E2 -9258.001} C_VEL
LIN {X 0,Y 439.481,Z 721.741,A -85,B 0,C 180,E1 -9261.725,E2 -9261.725} C_VEL
LIN {X 0,Y 439.599,Z 721.725,A -85,B 0,C 180,E1 -9264.496,E2 -9264.496} C_VEL
LIN {X 0,Y 439.628,Z 721.722,A -85,B 0,C 180,E1 -9268.168,E2 -9268.168} C_VEL
LIN {X 0,Y 439.672,Z 721.716,A -85,B 0,C 180,E1 -9270,E2 -9270} C_VEL
LIN {X 0,Y 439.505,Z 721.736,A -85,B 0,C 180,E1 -9270.97,E2 -9270.97} C_VEL
LIN {X 0,Y 438.861,Z 721.82,A -85,B 0,C 180,E1 -9271.735,E2 -9271.735} C_VEL
LIN {X 0,Y 435.924,Z 722.183,A -85,B 0,C 180,E1 -9272.975,E2 -9272.975} C_VEL
LIN {X 0,Y 433.463,Z 722.49,A -85,B 0,C 180,E1 -9273.976,E2 -9273.976} C_VEL
LIN {X 0,Y 432.479,Z 722.612,A -85,B 0,C 180,E1 -9274.752,E2 -9274.752} C_VEL
LIN {X 0,Y 432.441,Z 722.617,A -85,B 0,C 180,E1 -9275.014,E2 -9275.014} C_VEL
LIN {X 0,Y 432.517,Z 722.612,A -85,B 0,C 180,E1 -9277.607,E2 -9277.607} C_VEL
LIN {X 0,Y 432.393,Z 722.623,A -85,B 0,C 180,E1 -9281.248,E2 -9281.248} C_VEL
LIN {X 0,Y 432.376,Z 722.626,A -85,B 0,C 180,E1 -9284.112,E2 -9284.112} C_VEL
LIN {X 0,Y 432.398,Z 722.621,A -85,B 0,C 180,E1 -9287.012,E2 -9287.012} C_VEL
LIN {X 0,Y 432.343,Z 722.633,A -85,B 0,C 180,E1 -9289.96,E2 -9289.96} C_VEL
LIN {X 0,Y 432.32,Z 722.63,A -85,B 0,C 180,E1 -9292.964,E2 -9292.964} C_VEL
LIN {X 0,Y 432.338,Z 722.628,A -85,B 0,C 180,E1 -9295.002,E2 -9295.002} C_VEL
LIN {X 0,Y 432.35,Z 722.632,A -85,B 0,C 180,E1 -9298.126,E2 -9298.126} C_VEL
LIN {X 0,Y 432.324,Z 722.63,A -85,B 0,C 180,E1 -9301.346,E2 -9301.346} C_VEL
LIN {X 0,Y 432.341,Z 722.629,A -85,B 0,C 180,E1 -9304.677,E2 -9304.677} C_VEL
LIN {X 0,Y 432.339,Z 722.632,A -85,B 0,C 180,E1 -9308.15,E2 -9308.15} C_VEL
LIN {X 0,Y 432.336,Z 722.628,A -85,B 0,C 180,E1 -9311.602,E2 -9311.602} C_VEL
LIN {X 0,Y 432.337,Z 722.633,A -85,B 0,C 180,E1 -9314.347,E2 -9314.347} C_VEL
LIN {X 0,Y 432.38,Z 722.794,A -85,B 0,C 180,E1 -9316.413,E2 -9316.413} C_VEL
LIN {X 0,Y 435.31,Z 733.026,A -85,B 0,C 180,E1 -9317.113,E2 -9317.113} C_VEL
LIN {X 0,Y 435.836,Z 735.022,A -85,B 0,C 180,E1 -9317.266,E2 -9317.266} C_VEL
LIN {X 0,Y 435.422,Z 747.522,A -85,B 0,C 180,E1 -9318.208,E2 -9318.208} C_VEL
LIN {X 0,Y 434.911,Z 757.776,A -85,B 0,C 180,E1 -9319.178,E2 -9319.178} C_VEL
LIN {X 0,Y 434.389,Z 768.334,A -85,B 0,C 180,E1 -9320.427,E2 -9320.427} C_VEL
LIN {X 0,Y 433.86,Z 777.166,A -85,B 0,C 180,E1 -9321.713,E2 -9321.713} C_VEL
LIN {X 0,Y 433.385,Z 784.986,A -85,B 0,C 180,E1 -9323.129,E2 -9323.129} C_VEL
LIN {X 0,Y 432.987,Z 791.2,A -85,B 0,C 180,E1 -9324.53,E2 -9324.53} C_VEL
LIN {X 0,Y 432.675,Z 796.163,A -85,B 0,C 180,E1 -9325.935,E2 -9325.935} C_VEL
LIN {X 0,Y 432.499,Z 800.765,A -85,B 0,C 180,E1 -9327.671,E2 -9327.671} C_VEL
LIN {X 0,Y 432.292,Z 803.92,A -85,B 0,C 180,E1 -9329.503,E2 -9329.503} C_VEL
LIN {X 0,Y 432.23,Z 805.576,A -85,B 0,C 180,E1 -9331.407,E2 -9331.407} C_VEL
LIN {X 0,Y 432.285,Z 805.502,A -85,B 0,C 180,E1 -9333.404,E2 -9333.404} C_VEL
LIN {X 0,Y 432.445,Z 804.145,A -85,B 0,C 180,E1 -9335.004,E2 -9335.004} C_VEL
LIN {X 0,Y 432.669,Z 801.674,A -85,B 0,C 180,E1 -9336.549,E2 -9336.549} C_VEL
LIN {X 0,Y 432.951,Z 798.038,A -85,B 0,C 180,E1 -9338.077,E2 -9338.077} C_VEL
LIN {X 0,Y 433.339,Z 793.149,A -85,B 0,C 180,E1 -9339.592,E2 -9339.592} C_VEL
LIN {X 0,Y 433.787,Z 786.911,A -85,B 0,C 180,E1 -9341.093,E2 -9341.093} C_VEL
LIN {X 0,Y 434.372,Z 779.801,A -85,B 0,C 180,E1 -9342.446,E2 -9342.446} C_VEL
LIN {X 0,Y 434.969,Z 770.798,A -85,B 0,C 180,E1 -9343.816,E2 -9343.816} C_VEL
LIN {X 0,Y 435.588,Z 760.814,A -85,B 0,C 180,E1 -9345.039,E2 -9345.039} C_VEL
LIN {X 0,Y 436.12,Z 750.907,A -85,B 0,C 180,E1 -9346.012,E2 -9346.012} C_VEL
LIN {X 0,Y 436.532,Z 740.256,A -85,B 0,C 180,E1 -9346.855,E2 -9346.855} C_VEL
LIN {X 0,Y 436.615,Z 736.803,A -85,B 0,C 180,E1 -9347.095,E2 -9347.095} C_VEL
LIN {X 0,Y 433.672,Z 726.72,A -85,B 0,C 180,E1 -9347.838,E2 -9347.838} C_VEL
LIN {X 0,Y 432.448,Z 722.623,A -85,B 0,C 180,E1 -9348.13,E2 -9348.13} C_VEL
LIN {X 0,Y 432.468,Z 722.619,A -85,B 0,C 180,E1 -9351.59,E2 -9351.59} C_VEL
LIN {X 0,Y 432.585,Z 722.598,A -85,B 0,C 180,E1 -9354.406,E2 -9354.406} C_VEL
LIN {X 0,Y 432.606,Z 722.599,A -85,B 0,C 180,E1 -9358.138,E2 -9358.138} C_VEL
LIN {X 0,Y 432.732,Z 722.584,A -85,B 0,C 180,E1 -9360,E2 -9360} C_VEL
LIN {X 0,Y 432.588,Z 722.593,A -85,B 0,C 180,E1 -9362.794,E2 -9362.794} C_VEL
LIN {X 0,Y 432.564,Z 722.601,A -85,B 0,C 180,E1 -9366.53,E2 -9366.53} C_VEL
LIN {X 0,Y 432.443,Z 722.611,A -85,B 0,C 180,E1 -9369.353,E2 -9369.353} C_VEL
LIN {X 0,Y 432.435,Z 722.616,A -85,B 0,C 180,E1 -9372.803,E2 -9372.803} C_VEL
LIN {X 0,Y 432.416,Z 722.622,A -85,B 0,C 180,E1 -9376.479,E2 -9376.479} C_VEL
LIN {X 0,Y 432.343,Z 722.633,A -85,B 0,C 180,E1 -9379.96,E2 -9379.96} C_VEL
LIN {X 0,Y 432.321,Z 722.63,A -85,B 0,C 180,E1 -9382.964,E2 -9382.964} C_VEL
LIN {X 0,Y 432.364,Z 722.628,A -85,B 0,C 180,E1 -9386.032,E2 -9386.032} C_VEL
LIN {X 0,Y 432.346,Z 722.627,A -85,B 0,C 180,E1 -9389.187,E2 -9389.187} C_VEL
LIN {X 0,Y 432.326,Z 722.635,A -85,B 0,C 180,E1 -9392.443,E2 -9392.443} C_VEL
LIN {X 0,Y 432.347,Z 722.629,A -85,B 0,C 180,E1 -9395.632,E2 -9395.632} C_VEL
LIN {X 0,Y 432.353,Z 722.632,A -85,B 0,C 180,E1 -9399.343,E2 -9399.343} C_VEL
LIN {X 0,Y 432.336,Z 722.633,A -85,B 0,C 180,E1 -9401.797,E2 -9401.797} C_VEL
LIN {X 0,Y 432.336,Z 722.634,A -85,B 0,C 180,E1 -9404.347,E2 -9404.347} C_VEL
LIN {X 0,Y 432.379,Z 722.67,A -85,B 0,C 180,E1 -9407.692,E2 -9407.692} C_VEL
LIN {X 0,Y 433.857,Z 729.952,A -85,B 0,C 180,E1 -9410.25,E2 -9410.25} C_VEL
LIN {X 0,Y 435.296,Z 737.959,A -85,B 0,C 180,E1 -9412.84,E2 -9412.84} C_VEL
LIN {X 0,Y 435.253,Z 742.374,A -85,B 0,C 180,E1 -9414.133,E2 -9414.133} C_VEL
LIN {X 0,Y 434.567,Z 753.583,A -85,B 0,C 180,E1 -9417.242,E2 -9417.242} C_VEL
LIN {X 0,Y 433.861,Z 765.513,A -85,B 0,C 180,E1 -9420.392,E2 -9420.392} C_VEL
LIN {X 0,Y 433.368,Z 777.948,A -85,B 0,C 180,E1 -9423.564,E2 -9423.564} C_VEL
LIN {X 0,Y 432.815,Z 792.129,A -85,B 0,C 180,E1 -9427.063,E2 -9427.063} C_VEL
LIN {X 0,Y 432.429,Z 804.469,A -85,B 0,C 180,E1 -9430.044,E2 -9430.044} C_VEL
LIN {X 0,Y 432.179,Z 815.761,A -85,B 0,C 180,E1 -9432.736,E2 -9432.736} C_VEL
LIN {X 0,Y 432.108,Z 818.092,A -85,B 0,C 180,E1 -9433.228,E2 -9433.228} C_VEL
LIN {X 0,Y 433.434,Z 831.342,A -85,B 0,C 180,E1 -9433.638,E2 -9433.638} C_VEL
LIN {X 0,Y 434.264,Z 843.261,A -85,B 0,C 180,E1 -9434.151,E2 -9434.151} C_VEL
LIN {X 0,Y 435.025,Z 850.403,A -85,B 0,C 180,E1 -9434.54,E2 -9434.54} C_VEL
LIN {X 0,Y 434.406,Z 861.726,A -85,B 0,C 180,E1 -9435.237,E2 -9435.237} C_VEL
LIN {X 0,Y 433.655,Z 873.824,A -85,B 0,C 180,E1 -9436.194,E2 -9436.194} C_VEL
LIN {X 0,Y 433.171,Z 883.22,A -85,B 0,C 180,E1 -9437.109,E2 -9437.109} C_VEL
LIN {X 0,Y 432.631,Z 893.18,A -85,B 0,C 180,E1 -9438.284,E2 -9438.284} C_VEL
LIN {X 0,Y 432.203,Z 901.413,A -85,B 0,C 180,E1 -9439.459,E2 -9439.459} C_VEL
LIN {X 0,Y 431.888,Z 909.51,A -85,B 0,C 180,E1 -9440.871,E2 -9440.871} C_VEL
LIN {X 0,Y 431.702,Z 917,A -85,B 0,C 180,E1 -9442.517,E2 -9442.517} C_VEL
LIN {X 0,Y 431.659,Z 922.021,A -85,B 0,C 180,E1 -9443.925,E2 -9443.925} C_VEL
LIN {X 0,Y 431.641,Z 925.876,A -85,B 0,C 180,E1 -9445.33,E2 -9445.33} C_VEL
LIN {X 0,Y 431.662,Z 927.881,A -85,B 0,C 180,E1 -9446.266,E2 -9446.266} C_VEL
LIN {X 0,Y 431.619,Z 929.384,A -85,B 0,C 180,E1 -9447.2,E2 -9447.2} C_VEL
LIN {X 0,Y 431.621,Z 930.475,A -85,B 0,C 180,E1 -9448.134,E2 -9448.134} C_VEL
LIN {X 0,Y 431.603,Z 931.16,A -85,B 0,C 180,E1 -9449.067,E2 -9449.067} C_VEL
LIN {X 0,Y 431.598,Z 931.427,A -85,B 0,C 180,E1 -9450,E2 -9450} C_VEL
LIN {X 0,Y 431.592,Z 931.241,A -85,B 0,C 180,E1 -9450.933,E2 -9450.933} C_VEL
LIN {X 0,Y 431.6,Z 930.651,A -85,B 0,C 180,E1 -9451.866,E2 -9451.866} C_VEL
LIN {X 0,Y 431.596,Z 929.656,A -85,B 0,C 180,E1 -9452.8,E2 -9452.8} C_VEL
LIN {X 0,Y 431.659,Z 928.238,A -85,B 0,C 180,E1 -9453.734,E2 -9453.734} C_VEL
LIN {X 0,Y 431.584,Z 925.224,A -85,B 0,C 180,E1 -9455.138,E2 -9455.138} C_VEL
LIN {X 0,Y 431.582,Z 920.898,A -85,B 0,C 180,E1 -9456.614,E2 -9456.614} C_VEL
LIN {X 0,Y 431.745,Z 914.839,A -85,B 0,C 180,E1 -9458.189,E2 -9458.189} C_VEL
LIN {X 0,Y 431.973,Z 907.981,A -85,B 0,C 180,E1 -9459.6,E2 -9459.6} C_VEL
LIN {X 0,Y 432.366,Z 899.488,A -85,B 0,C 180,E1 -9461.011,E2 -9461.011} C_VEL
LIN {X 0,Y 432.848,Z 890.764,A -85,B 0,C 180,E1 -9462.185,E2 -9462.185} C_VEL
LIN {X 0,Y 433.372,Z 881.601,A -85,B 0,C 180,E1 -9463.206,E2 -9463.206} C_VEL
LIN {X 0,Y 434.039,Z 869.504,A -85,B 0,C 180,E1 -9464.296,E2 -9464.296} C_VEL
LIN {X 0,Y 434.808,Z 857.915,A -85,B 0,C 180,E1 -9465.108,E2 -9465.108} C_VEL
LIN {X 0,Y 435.047,Z 849.588,A -85,B 0,C 180,E1 -9465.579,E2 -9465.579} C_VEL
LIN {X 0,Y 433.822,Z 837.131,A -85,B 0,C 180,E1 -9466.177,E2 -9466.177} C_VEL
LIN {X 0,Y 432.486,Z 824.21,A -85,B 0,C 180,E1 -9466.613,E2 -9466.613} C_VEL
LIN {X 0,Y 432.141,Z 820.629,A -85,B 0,C 180,E1 -9466.715,E2 -9466.715} C_VEL
LIN {X 0,Y 432.476,Z 809.235,A -85,B 0,C 180,E1 -9469.518,E2 -9469.518} C_VEL
LIN {X 0,Y 433.04,Z 795.55,A -85,B 0,C 180,E1 -9472.924,E2 -9472.924} C_VEL
LIN {X 0,Y 433.74,Z 781.569,A -85,B 0,C 180,E1 -9476.461,E2 -9476.461} C_VEL
LIN {X 0,Y 434.493,Z 767.568,A -85,B 0,C 180,E1 -9480.095,E2 -9480.095} C_VEL
LIN {X 0,Y 435.315,Z 755.527,A -85,B 0,C 180,E1 -9483.293,E2 -9483.293} C_VEL
LIN {X 0,Y 436.097,Z 744.51,A -85,B 0,C 180,E1 -9486.314,E2 -9486.314} C_VEL
LIN {X 0,Y 435.983,Z 740.424,A -85,B 0,C 180,E1 -9487.478,E2 -9487.478} C_VEL
LIN {X 0,Y 433.603,Z 728.753,A -85,B 0,C 180,E1 -9491.09,E2 -9491.09} C_VEL
LIN {X 0,Y 432.341,Z 722.633,A -85,B 0,C 180,E1 -9493.138,E2 -9493.138} C_VEL
LIN {X 0,Y 432.335,Z 722.632,A -85,B 0,C 180,E1 -9495.665,E2 -9495.665} C_VEL
LIN {X 0,Y 432.334,Z 722.63,A -85,B 0,C 180,E1 -9498.398,E2 -9498.398} C_VEL
LIN {X 0,Y 432.339,Z 722.63,A -85,B 0,C 180,E1 -9501.85,E2 -9501.85} C_VEL
LIN {X 0,Y 432.342,Z 722.63,A -85,B 0,C 180,E1 -9505.323,E2 -9505.323} C_VEL
LIN {X 0,Y 432.323,Z 722.63,A -85,B 0,C 180,E1 -9508.654,E2 -9508.654} C_VEL
LIN {X 0,Y 432.384,Z 722.627,A -85,B 0,C 180,E1 -9511.877,E2 -9511.877} C_VEL
LIN {X 0,Y 432.348,Z 722.627,A -85,B 0,C 180,E1 -9514.999,E2 -9514.999} C_VEL
LIN {X 0,Y 432.36,Z 722.63,A -85,B 0,C 180,E1 -9518.046,E2 -9518.046} C_VEL
LIN {X 0,Y 432.387,Z 722.623,A -85,B 0,C 180,E1 -9521.03,E2 -9521.03} C_VEL
LIN {X 0,Y 432.433,Z 722.622,A -85,B 0,C 180,E1 -9523.961,E2 -9523.961} C_VEL
LIN {X 0,Y 432.462,Z 722.616,A -85,B 0,C 180,E1 -9527.804,E2 -9527.804} C_VEL
LIN {X 0,Y 432.494,Z 722.61,A -85,B 0,C 180,E1 -9531.59,E2 -9531.59} C_VEL
LIN {X 0,Y 432.597,Z 722.6,A -85,B 0,C 180,E1 -9534.406,E2 -9534.406} C_VEL
LIN {X 0,Y 432.603,Z 722.599,A -85,B 0,C 180,E1 -9538.138,E2 -9538.138} C_VEL
LIN {X 0,Y 432.731,Z 722.582,A -85,B 0,C 180,E1 -9540,E2 -9540} C_VEL
LIN {X 0,Y 432.586,Z 722.6,A -85,B 0,C 180,E1 -9542.794,E2 -9542.794} C_VEL
LIN {X 0,Y 432.585,Z 722.6,A -85,B 0,C 180,E1 -9545.594,E2 -9545.594} C_VEL
LIN {X 0,Y 432.466,Z 722.616,A -85,B 0,C 180,E1 -9548.41,E2 -9548.41} C_VEL
LIN {X 0,Y 432.462,Z 722.615,A -85,B 0,C 180,E1 -9552.197,E2 -9552.197} C_VEL
LIN {X 0,Y 432.432,Z 722.619,A -85,B 0,C 180,E1 -9556.039,E2 -9556.039} C_VEL
LIN {X 0,Y 432.389,Z 722.624,A -85,B 0,C 180,E1 -9559.485,E2 -9559.485} C_VEL
LIN {X 0,Y 432.313,Z 722.636,A -85,B 0,C 180,E1 -9562.965,E2 -9562.965} C_VEL
LIN {X 0,Y 432.321,Z 722.634,A -85,B 0,C 180,E1 -9566.035,E2 -9566.035} C_VEL
LIN {X 0,Y 432.334,Z 722.632,A -85,B 0,C 180,E1 -9569.188,E2 -9569.188} C_VEL
LIN {X 0,Y 432.323,Z 722.633,A -85,B 0,C 180,E1 -9572.443,E2 -9572.443} C_VEL
LIN {X 0,Y 432.337,Z 722.63,A -85,B 0,C 180,E1 -9575.818,E2 -9575.818} C_VEL
LIN {X 0,Y 432.302,Z 722.636,A -85,B 0,C 180,E1 -9579.348,E2 -9579.348} C_VEL
LIN {X 0,Y 432.305,Z 722.634,A -85,B 0,C 180,E1 -9581.801,E2 -9581.801} C_VEL
LIN {X 0,Y 432.333,Z 722.632,A -85,B 0,C 180,E1 -9584.348,E2 -9584.348} C_VEL
LIN {X 0,Y 432.304,Z 722.635,A -85,B 0,C 180,E1 -9587.018,E2 -9587.018} C_VEL
LIN {X 0,Y 432.29,Z 722.636,A -85,B 0,C 180,E1 -9589.828,E2 -9589.828} C_VEL
LIN {X 0,Y 432.298,Z 722.636,A -85,B 0,C 180,E1 -9593.021,E2 -9593.021} C_VEL
LIN {X 0,Y 432.332,Z 722.631,A -85,B 0,C 180,E1 -9596.003,E2 -9596.003} C_VEL
LIN {X 0,Y 432.339,Z 722.631,A -85,B 0,C 180,E1 -9599.492,E2 -9599.492} C_VEL
LIN {X 0,Y 432.316,Z 722.634,A -85,B 0,C 180,E1 -9601.872,E2 -9601.872} C_VEL
LIN {X 0,Y 432.35,Z 722.629,A -85,B 0,C 180,E1 -9605.548,E2 -9605.548} C_VEL
LIN {X 0,Y 432.353,Z 722.631,A -85,B 0,C 180,E1 -9609.046,E2 -9609.046} C_VEL
LIN {X 0,Y 432.36,Z 722.628,A -85,B 0,C 180,E1 -9612.01,E2 -9612.01} C_VEL
LIN {X 0,Y 432.389,Z 722.625,A -85,B 0,C 180,E1 -9614.926,E2 -9614.926} C_VEL
LIN {X 0,Y 432.456,Z 722.615,A -85,B 0,C 180,E1 -9617.803,E2 -9617.803} C_VEL
LIN {X 0,Y 432.448,Z 722.617,A -85,B 0,C 180,E1 -9621.59,E2 -9621.59} C_VEL
LIN {X 0,Y 432.554,Z 722.603,A -85,B 0,C 180,E1 -9624.406,E2 -9624.406} C_VEL
LIN {X 0,Y 432.598,Z 722.597,A -85,B 0,C 180,E1 -9628.138,E2 -9628.138} C_VEL
LIN {X 0,Y 432.623,Z 722.594,A -85,B 0,C 180,E1 -9630,E2 -9630} C_VEL
LIN {X 0,Y 432.562,Z 722.601,A -85,B 0,C 180,E1 -9632.794,E2 -9632.794} C_VEL
LIN {X 0,Y 432.441,Z 722.617,A -85,B 0,C 180,E1 -9635.014,E2 -9635.014} C_VEL
LIN {X 0,Y 431.876,Z 722.69,A -85,B 0,C 180,E1 -9635.793,E2 -9635.793} C_VEL
LIN {X 0,Y 429.022,Z 723.043,A -85,B 0,C 180,E1 -9637.057,E2 -9637.057} C_VEL
LIN {X 0,Y 426.541,Z 723.352,A -85,B 0,C 180,E1 -9638.077,E2 -9638.077} C_VEL
LIN {X 0,Y 425.473,Z 723.484,A -85,B 0,C 180,E1 -9638.867,E2 -9638.867} C_VEL
LIN {X 0,Y 425.388,Z 723.495,A -85,B 0,C 180,E1 -9639.135,E2 -9639.135} C_VEL
LIN {X 0,Y 425.397,Z 723.493,A -85,B 0,C 180,E1 -9642.904,E2 -9642.904} C_VEL
LIN {X 0,Y 425.364,Z 723.497,A -85,B 0,C 180,E1 -9646.605,E2 -9646.605} C_VEL
LIN {X 0,Y 425.332,Z 723.504,A -85,B 0,C 180,E1 -9649.636,E2 -9649.636} C_VEL
LIN {X 0,Y 425.291,Z 723.508,A -85,B 0,C 180,E1 -9652.339,E2 -9652.339} C_VEL
LIN {X 0,Y 425.321,Z 723.503,A -85,B 0,C 180,E1 -9654.656,E2 -9654.656} C_VEL
LIN {X 0,Y 425.274,Z 723.509,A -85,B 0,C 180,E1 -9657.563,E2 -9657.563} C_VEL
LIN {X 0,Y 425.294,Z 723.506,A -85,B 0,C 180,E1 -9660.761,E2 -9660.761} C_VEL
LIN {X 0,Y 425.313,Z 723.508,A -85,B 0,C 180,E1 -9664.288,E2 -9664.288} C_VEL
LIN {X 0,Y 425.282,Z 723.507,A -85,B 0,C 180,E1 -9667.694,E2 -9667.694} C_VEL
LIN {X 0,Y 425.283,Z 723.511,A -85,B 0,C 180,E1 -9670.52,E2 -9670.52} C_VEL
LIN {X 0,Y 425.26,Z 723.509,A -85,B 0,C 180,E1 -9673.351,E2 -9673.351} C_VEL
LIN {X 0,Y 425.294,Z 723.509,A -85,B 0,C 180,E1 -9676.159,E2 -9676.159} C_VEL
LIN {X 0,Y 428.701,Z 735.443,A -85,B 0,C 180,E1 -9677.004,E2 -9677.004} C_VEL
LIN {X 0,Y 429.002,Z 738.448,A -85,B 0,C 180,E1 -9677.227,E2 -9677.227} C_VEL
LIN {X 0,Y 428.516,Z 749.09,A -85,B 0,C 180,E1 -9678.061,E2 -9678.061} C_VEL
LIN {X 0,Y 427.948,Z 760.2,A -85,B 0,C 180,E1 -9679.158,E2 -9679.158} C_VEL
LIN {X 0,Y 427.379,Z 770.526,A -85,B 0,C 180,E1 -9680.425,E2 -9680.425} C_VEL
LIN {X 0,Y 426.78,Z 779.603,A -85,B 0,C 180,E1 -9681.816,E2 -9681.816} C_VEL
LIN {X 0,Y 426.338,Z 787.382,A -85,B 0,C 180,E1 -9683.304,E2 -9683.304} C_VEL
LIN {X 0,Y 425.935,Z 793.34,A -85,B 0,C 180,E1 -9684.724,E2 -9684.724} C_VEL
LIN {X 0,Y 425.612,Z 798.796,A -85,B 0,C 180,E1 -9686.415,E2 -9686.415} C_VEL
LIN {X 0,Y 425.437,Z 802.711,A -85,B 0,C 180,E1 -9688.087,E2 -9688.087} C_VEL
LIN {X 0,Y 425.294,Z 804.64,A -85,B 0,C 180,E1 -9689.239,E2 -9689.239} C_VEL
LIN {X 0,Y 425.203,Z 806.492,A -85,B 0,C 180,E1 -9691.166,E2 -9691.166} C_VEL
LIN {X 0,Y 425.205,Z 806.804,A -85,B 0,C 180,E1 -9692.432,E2 -9692.432} C_VEL
LIN {X 0,Y 425.277,Z 806.539,A -85,B 0,C 180,E1 -9693.5,E2 -9693.5} C_VEL
LIN {X 0,Y 425.485,Z 804.912,A -85,B 0,C 180,E1 -9695.295,E2 -9695.295} C_VEL
LIN {X 0,Y 425.709,Z 802.715,A -85,B 0,C 180,E1 -9696.658,E2 -9696.658} C_VEL
LIN {X 0,Y 425.994,Z 799.088,A -85,B 0,C 180,E1 -9698.21,E2 -9698.21} C_VEL
LIN {X 0,Y 426.476,Z 793.522,A -85,B 0,C 180,E1 -9699.938,E2 -9699.938} C_VEL
LIN {X 0,Y 426.913,Z 787.95,A -85,B 0,C 180,E1 -9701.275,E2 -9701.275} C_VEL
LIN {X 0,Y 427.454,Z 781.77,A -85,B 0,C 180,E1 -9702.481,E2 -9702.481} C_VEL
LIN {X 0,Y 428.043,Z 773.598,A -85,B 0,C 180,E1 -9703.792,E2 -9703.792} C_VEL
LIN {X 0,Y 428.622,Z 764.687,A -85,B 0,C 180,E1 -9704.951,E2 -9704.951} C_VEL
LIN {X 0,Y 429.226,Z 754.525,A -85,B 0,C 180,E1 -9706.024,E2 -9706.024} C_VEL
LIN {X 0,Y 429.655,Z 744.531,A -85,B 0,C 180,E1 -9706.882,E2 -9706.882} C_VEL
LIN {X 0,Y 429.782,Z 737.867,A -85,B 0,C 180,E1 -9707.366,E2 -9707.366} C_VEL
LIN {X 0,Y 426.298,Z 726.456,A -85,B 0,C 180,E1 -9708.228,E2 -9708.228} C_VEL
LIN {X 0,Y 425.372,Z 723.503,A -85,B 0,C 180,E1 -9708.444,E2 -9708.444} C_VEL
LIN {X 0,Y 425.412,Z 723.497,A -85,B 0,C 180,E1 -9711.449,E2 -9711.449} C_VEL
LIN {X 0,Y 425.54,Z 723.475,A -85,B 0,C 180,E1 -9714.313,E2 -9714.313} C_VEL
LIN {X 0,Y 425.575,Z 723.475,A -85,B 0,C 180,E1 -9718.107,E2 -9718.107} C_VEL
LIN {X 0,Y 425.701,Z 723.459,A -85,B 0,C 180,E1 -9720,E2 -9720} C_VEL
LIN {X 0,Y 425.542,Z 723.471,A -85,B 0,C 180,E1 -9722.84,E2 -9722.84} C_VEL
LIN {X 0,Y 425.553,Z 723.474,A -85,B 0,C 180,E1 -9725.687,E2 -9725.687} C_VEL
LIN {X 0,Y 425.439,Z 723.484,A -85,B 0,C 180,E1 -9728.55,E2 -9728.55} C_VEL
LIN {X 0,Y 425.416,Z 723.492,A -85,B 0,C 180,E1 -9732.402,E2 -9732.402} C_VEL
LIN {X 0,Y 425.392,Z 723.499,A -85,B 0,C 180,E1 -9736.312,E2 -9736.312} C_VEL
LIN {X 0,Y 425.332,Z 723.503,A -85,B 0,C 180,E1 -9739.635,E2 -9739.635} C_VEL
LIN {X 0,Y 425.291,Z 723.512,A -85,B 0,C 180,E1 -9742.339,E2 -9742.339} C_VEL
LIN {X 0,Y 425.294,Z 723.506,A -85,B 0,C 180,E1 -9745.445,E2 -9745.445} C_VEL
LIN {X 0,Y 425.352,Z 723.499,A -85,B 0,C 180,E1 -9747.557,E2 -9747.557} C_VEL
LIN {X 0,Y 425.291,Z 723.507,A -85,B 0,C 180,E1 -9750.816,E2 -9750.816} C_VEL
LIN {X 0,Y 425.315,Z 723.509,A -85,B 0,C 180,E1 -9754.288,E2 -9754.288} C_VEL
LIN {X 0,Y 425.283,Z 723.512,A -85,B 0,C 180,E1 -9757.694,E2 -9757.694} C_VEL
LIN {X 0,Y 425.284,Z 723.514,A -85,B 0,C 180,E1 -9760.52,E2 -9760.52} C_VEL
LIN {X 0,Y 425.26,Z 723.514,A -85,B 0,C 180,E1 -9763.351,E2 -9763.351} C_VEL
LIN {X 0,Y 425.26,Z 723.516,A -85,B 0,C 180,E1 -9766.649,E2 -9766.649} C_VEL
LIN {X 0,Y 425.298,Z 723.557,A -85,B 0,C 180,E1 -9767.279,E2 -9767.279} C_VEL
LIN {X 0,Y 426.88,Z 731.193,A -85,B 0,C 180,E1 -9770.052,E2 -9770.052} C_VEL
LIN {X 0,Y 428.3,Z 738.937,A -85,B 0,C 180,E1 -9772.617,E2 -9772.617} C_VEL
LIN {X 0,Y 428.401,Z 742.811,A -85,B 0,C 180,E1 -9773.801,E2 -9773.801} C_VEL
LIN {X 0,Y 427.577,Z 754.626,A -85,B 0,C 180,E1 -9777.152,E2 -9777.152} C_VEL
LIN {X 0,Y 426.869,Z 765.64,A -85,B 0,C 180,E1 -9780.129,E2 -9780.129} C_VEL
LIN {X 0,Y 426.298,Z 778.846,A -85,B 0,C 180,E1 -9783.568,E2 -9783.568} C_VEL
LIN {X 0,Y 425.749,Z 792.136,A -85,B 0,C 180,E1 -9786.918,E2 -9786.918} C_VEL
LIN {X 0,Y 425.336,Z 805.034,A -85,B 0,C 180,E1 -9790.097,E2 -9790.097} C_VEL
LIN {X 0,Y 425.072,Z 816.53,A -85,B 0,C 180,E1 -9792.893,E2 -9792.893} C_VEL
LIN {X 0,Y 426.584,Z 832.387,A -85,B 0,C 180,E1 -9793.432,E2 -9793.432} C_VEL
LIN {X 0,Y 427.426,Z 844.883,A -85,B 0,C 180,E1 -9794.013,E2 -9794.013} C_VEL
LIN {X 0,Y 428.018,Z 851.517,A -85,B 0,C 180,E1 -9794.402,E2 -9794.402} C_VEL
LIN {X 0,Y 427.258,Z 863.92,A -85,B 0,C 180,E1 -9795.229,E2 -9795.229} C_VEL
LIN {X 0,Y 426.57,Z 875.662,A -85,B 0,C 180,E1 -9796.227,E2 -9796.227} C_VEL
LIN {X 0,Y 426.1,Z 884.548,A -85,B 0,C 180,E1 -9797.154,E2 -9797.154} C_VEL
LIN {X 0,Y 425.534,Z 893.894,A -85,B 0,C 180,E1 -9798.327,E2 -9798.327} C_VEL
LIN {X 0,Y 425.036,Z 903.215,A -85,B 0,C 180,E1 -9799.761,E2 -9799.761} C_VEL
LIN {X 0,Y 424.755,Z 910.785,A -85,B 0,C 180,E1 -9801.196,E2 -9801.196} C_VEL
LIN {X 0,Y 424.642,Z 915.929,A -85,B 0,C 180,E1 -9802.391,E2 -9802.391} C_VEL
LIN {X 0,Y 424.603,Z 921.377,A -85,B 0,C 180,E1 -9803.953,E2 -9803.953} C_VEL
LIN {X 0,Y 424.604,Z 924.837,A -85,B 0,C 180,E1 -9805.253,E2 -9805.253} C_VEL
LIN {X 0,Y 424.627,Z 926.847,A -85,B 0,C 180,E1 -9806.204,E2 -9806.204} C_VEL
LIN {X 0,Y 424.58,Z 928.355,A -85,B 0,C 180,E1 -9807.153,E2 -9807.153} C_VEL
LIN {X 0,Y 424.585,Z 929.456,A -85,B 0,C 180,E1 -9808.103,E2 -9808.103} C_VEL
LIN {X 0,Y 424.573,Z 930.147,A -85,B 0,C 180,E1 -9809.051,E2 -9809.051} C_VEL
LIN {X 0,Y 424.57,Z 930.416,A -85,B 0,C 180,E1 -9810,E2 -9810} C_VEL
LIN {X 0,Y 424.562,Z 930.231,A -85,B 0,C 180,E1 -9810.948,E2 -9810.948} C_VEL
LIN {X 0,Y 424.563,Z 929.645,A -85,B 0,C 180,E1 -9811.897,E2 -9811.897} C_VEL
LIN {X 0,Y 424.557,Z 928.651,A -85,B 0,C 180,E1 -9812.846,E2 -9812.846} C_VEL
LIN {X 0,Y 424.624,Z 927.23,A -85,B 0,C 180,E1 -9813.796,E2 -9813.796} C_VEL
LIN {X 0,Y 424.533,Z 924.212,A -85,B 0,C 180,E1 -9815.224,E2 -9815.224} C_VEL
LIN {X 0,Y 424.541,Z 920.119,A -85,B 0,C 180,E1 -9816.654,E2 -9816.654} C_VEL
LIN {X 0,Y 424.703,Z 913.816,A -85,B 0,C 180,E1 -9818.325,E2 -9818.325} C_VEL
LIN {X 0,Y 424.915,Z 906.948,A -85,B 0,C 180,E1 -9819.761,E2 -9819.761} C_VEL
LIN {X 0,Y 425.35,Z 898.444,A -85,B 0,C 180,E1 -9821.195,E2 -9821.195} C_VEL
LIN {X 0,Y 425.88,Z 889.711,A -85,B 0,C 180,E1 -9822.388,E2 -9822.388} C_VEL
LIN {X 0,Y 426.489,Z 879.503,A -85,B 0,C 180,E1 -9823.53,E2 -9823.53} C_VEL
LIN {X 0,Y 427.111,Z 868.427,A -85,B 0,C 180,E1 -9824.533,E2 -9824.533} C_VEL
LIN {X 0,Y 427.909,Z 856.805,A -85,B 0,C 180,E1 -9825.357,E2 -9825.357} C_VEL
LIN {X 0,Y 428.006,Z 849.566,A -85,B 0,C 180,E1 -9825.781,E2 -9825.781} C_VEL
LIN {X 0,Y 426.82,Z 836.868,A -85,B 0,C 180,E1 -9826.409,E2 -9826.409} C_VEL
LIN {X 0,Y 425.57,Z 824.477,A -85,B 0,C 180,E1 -9826.849,E2 -9826.849} C_VEL
LIN {X 0,Y 425.09,Z 819.711,A -85,B 0,C 180,E1 -9826.991,E2 -9826.991} C_VEL
LIN {X 0,Y 425.537,Z 806.582,A -85,B 0,C 180,E1 -9830.293,E2 -9830.293} C_VEL
LIN {X 0,Y 426.135,Z 792.671,A -85,B 0,C 180,E1 -9833.833,E2 -9833.833} C_VEL
LIN {X 0,Y 426.908,Z 778.733,A -85,B 0,C 180,E1 -9837.449,E2 -9837.449} C_VEL
LIN {X 0,Y 427.774,Z 764.194,A -85,B 0,C 180,E1 -9841.315,E2 -9841.315} C_VEL
LIN {X 0,Y 428.632,Z 752.831,A -85,B 0,C 180,E1 -9844.427,E2 -9844.427} C_VEL
LIN {X 0,Y 429.252,Z 743.955,A -85,B 0,C 180,E1 -9846.908,E2 -9846.908} C_VEL
LIN {X 0,Y 428.349,Z 738.532,A -85,B 0,C 180,E1 -9848.57,E2 -9848.57} C_VEL
LIN {X 0,Y 426.387,Z 728.828,A -85,B 0,C 180,E1 -9851.649,E2 -9851.649} C_VEL
LIN {X 0,Y 425.283,Z 723.512,A -85,B 0,C 180,E1 -9853.487,E2 -9853.487} C_VEL
LIN {X 0,Y 425.259,Z 723.512,A -85,B 0,C 180,E1 -9856.649,E2 -9856.649} C_VEL
LIN {X 0,Y 425.288,Z 723.508,A -85,B 0,C 180,E1 -9859.873,E2 -9859.873} C_VEL
LIN {X 0,Y 425.28,Z 723.507,A -85,B 0,C 180,E1 -9862.488,E2 -9862.488} C_VEL
LIN {X 0,Y 425.309,Z 723.507,A -85,B 0,C 180,E1 -9865.817,E2 -9865.817} C_VEL
LIN {X 0,Y 425.292,Z 723.507,A -85,B 0,C 180,E1 -9869.239,E2 -9869.239} C_VEL
LIN {X 0,Y 425.35,Z 723.499,A -85,B 0,C 180,E1 -9872.442,E2 -9872.442} C_VEL
LIN {X 0,Y 425.35,Z 723.502,A -85,B 0,C 180,E1 -9875.602,E2 -9875.602} C_VEL
LIN {X 0,Y 425.295,Z 723.506,A -85,B 0,C 180,E1 -9878.682,E2 -9878.682} C_VEL
LIN {X 0,Y 425.332,Z 723.504,A -85,B 0,C 180,E1 -9881.703,E2 -9881.703} C_VEL
LIN {X 0,Y 425.35,Z 723.5,A -85,B 0,C 180,E1 -9884.671,E2 -9884.671} C_VEL
LIN {X 0,Y 425.414,Z 723.492,A -85,B 0,C 180,E1 -9887.598,E2 -9887.598} C_VEL
LIN {X 0,Y 425.445,Z 723.488,A -85,B 0,C 180,E1 -9891.45,E2 -9891.45} C_VEL
LIN {X 0,Y 425.553,Z 723.479,A -85,B 0,C 180,E1 -9894.313,E2 -9894.313} C_VEL
LIN {X 0,Y 425.572,Z 723.474,A -85,B 0,C 180,E1 -9898.107,E2 -9898.107} C_VEL
LIN {X 0,Y 425.7,Z 723.457,A -85,B 0,C 180,E1 -9900,E2 -9900} C_VEL
LIN {X 0,Y 425.539,Z 723.477,A -85,B 0,C 180,E1 -9902.84,E2 -9902.84} C_VEL
LIN {X 0,Y 425.498,Z 723.484,A -85,B 0,C 180,E1 -9906.529,E2 -9906.529} C_VEL
LIN {X 0,Y 425.4,Z 723.494,A -85,B 0,C 180,E1 -9909.51,E2 -9909.51} C_VEL
LIN {X 0,Y 425.396,Z 723.496,A -85,B 0,C 180,E1 -9912.904,E2 -9912.904} C_VEL
LIN {X 0,Y 425.363,Z 723.501,A -85,B 0,C 180,E1 -9916.605,E2 -9916.605} C_VEL
LIN {X 0,Y 425.331,Z 723.503,A -85,B 0,C 180,E1 -9919.636,E2 -9919.636} C_VEL
LIN {X 0,Y 425.289,Z 723.508,A -85,B 0,C 180,E1 -9922.339,E2 -9922.339} C_VEL
LIN {X 0,Y 425.261,Z 723.512,A -85,B 0,C 180,E1 -9925.448,E2 -9925.448} C_VEL
LIN {X 0,Y 425.314,Z 723.507,A -85,B 0,C 180,E1 -9928.862,E2 -9928.862} C_VEL
LIN {X 0,Y 425.265,Z 723.512,A -85,B 0,C 180,E1 -9931.927,E2 -9931.927} C_VEL
LIN {X 0,Y 425.296,Z 723.509,A -85,B 0,C 180,E1 -9935.337,E2 -9935.337} C_VEL
LIN {X 0,Y 425.279,Z 723.51,A -85,B 0,C 180,E1 -9938.901,E2 -9938.901} C_VEL
LIN {X 0,Y 425.258,Z 723.513,A -85,B 0,C 180,E1 -9942.656,E2 -9942.656} C_VEL
LIN {X 0,Y 425.285,Z 723.51,A -85,B 0,C 180,E1 -9945.284,E2 -9945.284} C_VEL
LIN {X 0,Y 425.249,Z 723.515,A -85,B 0,C 180,E1 -9948.618,E2 -9948.618} C_VEL
LIN {X 0,Y 425.278,Z 723.51,A -85,B 0,C 180,E1 -9951.099,E2 -9951.099} C_VEL
LIN {X 0,Y 425.293,Z 723.51,A -85,B 0,C 180,E1 -9954.663,E2 -9954.663} C_VEL
LIN {X 0,Y 425.248,Z 723.513,A -85,B 0,C 180,E1 -9958.072,E2 -9958.072} C_VEL
LIN {X 0,Y 425.297,Z 723.507,A -85,B 0,C 180,E1 -9961.365,E2 -9961.365} C_VEL
LIN {X 0,Y 425.253,Z 723.513,A -85,B 0,C 180,E1 -9964.552,E2 -9964.552} C_VEL
LIN {X 0,Y 425.294,Z 723.508,A -85,B 0,C 180,E1 -9967.73,E2 -9967.73} C_VEL
LIN {X 0,Y 425.364,Z 723.5,A -85,B 0,C 180,E1 -9970.704,E2 -9970.704} C_VEL
LIN {X 0,Y 425.388,Z 723.496,A -85,B 0,C 180,E1 -9973.688,E2 -9973.688} C_VEL
LIN {X 0,Y 425.411,Z 723.493,A -85,B 0,C 180,E1 -9977.598,E2 -9977.598} C_VEL
LIN {X 0,Y 425.396,Z 723.496,A -85,B 0,C 180,E1 -9981.449,E2 -9981.449} C_VEL
LIN {X 0,Y 425.512,Z 723.481,A -85,B 0,C 180,E1 -9984.313,E2 -9984.313} C_VEL
LIN {X 0,Y 425.567,Z 723.473,A -85,B 0,C 180,E1 -9988.107,E2 -9988.107} C_VEL
LIN {X 0,Y 425.576,Z 723.472,A -85,B 0,C 180,E1 -9990,E2 -9990} C_VEL
LIN {X 0,Y 425.517,Z 723.479,A -85,B 0,C 180,E1 -9992.84,E2 -9992.84} C_VEL
LIN {X 0,Y 425.53,Z 723.481,A -85,B 0,C 180,E1 -9995.687,E2 -9995.687} C_VEL
LIN {X 0,Y 425.41,Z 723.492,A -85,B 0,C 180,E1 -9998.551,E2 -9998.551} C_VEL
LIN {X 0,Y 425.388,Z 723.495,A -85,B 0,C 180,E1 -9999.135,E2 -9999.135} C_VEL
LIN {X 0,Y 424.733,Z 723.58,A -85,B 0,C 180,E1 -9999.925,E2 -9999.925} C_VEL
LIN {X 0,Y 421.895,Z 723.931,A -85,B 0,C 180,E1 -10001.208,E2 -10001.208} C_VEL
LIN {X 0,Y 419.476,Z 724.232,A -85,B 0,C 180,E1 -10002.245,E2 -10002.245} C_VEL
LIN {X 0,Y 418.421,Z 724.363,A -85,B 0,C 180,E1 -10003.046,E2 -10003.046} C_VEL
LIN {X 0,Y 418.327,Z 724.376,A -85,B 0,C 180,E1 -10003.317,E2 -10003.317} C_VEL
LIN {X 0,Y 418.316,Z 724.375,A -85,B 0,C 180,E1 -10006.735,E2 -10006.735} C_VEL
LIN {X 0,Y 418.274,Z 724.385,A -85,B 0,C 180,E1 -10009.79,E2 -10009.79} C_VEL
LIN {X 0,Y 418.235,Z 724.385,A -85,B 0,C 180,E1 -10012.737,E2 -10012.737} C_VEL
LIN {X 0,Y 418.237,Z 724.39,A -85,B 0,C 180,E1 -10015.907,E2 -10015.907} C_VEL
LIN {X 0,Y 418.264,Z 724.381,A -85,B 0,C 180,E1 -10019.162,E2 -10019.162} C_VEL
LIN {X 0,Y 418.261,Z 724.382,A -85,B 0,C 180,E1 -10022.844,E2 -10022.844} C_VEL
LIN {X 0,Y 418.248,Z 724.39,A -85,B 0,C 180,E1 -10026.238,E2 -10026.238} C_VEL
LIN {X 0,Y 418.248,Z 724.383,A -85,B 0,C 180,E1 -10029.683,E2 -10029.683} C_VEL
LIN {X 0,Y 418.233,Z 724.391,A -85,B 0,C 180,E1 -10032.321,E2 -10032.321} C_VEL
LIN {X 0,Y 418.241,Z 724.386,A -85,B 0,C 180,E1 -10035.916,E2 -10035.916} C_VEL
LIN {X 0,Y 421.545,Z 736.016,A -85,B 0,C 180,E1 -10036.748,E2 -10036.748} C_VEL
LIN {X 0,Y 422.185,Z 738.622,A -85,B 0,C 180,E1 -10036.959,E2 -10036.959} C_VEL
LIN {X 0,Y 421.643,Z 750.077,A -85,B 0,C 180,E1 -10037.864,E2 -10037.864} C_VEL
LIN {X 0,Y 421.046,Z 761.335,A -85,B 0,C 180,E1 -10038.995,E2 -10038.995} C_VEL
LIN {X 0,Y 420.461,Z 771.437,A -85,B 0,C 180,E1 -10040.255,E2 -10040.255} C_VEL
LIN {X 0,Y 419.97,Z 779.2,A -85,B 0,C 180,E1 -10041.438,E2 -10041.438} C_VEL
LIN {X 0,Y 419.441,Z 787.028,A -85,B 0,C 180,E1 -10042.9,E2 -10042.9} C_VEL
LIN {X 0,Y 419.036,Z 793.264,A -85,B 0,C 180,E1 -10044.35,E2 -10044.35} C_VEL
LIN {X 0,Y 418.66,Z 798.342,A -85,B 0,C 180,E1 -10045.836,E2 -10045.836} C_VEL
LIN {X 0,Y 418.483,Z 802.622,A -85,B 0,C 180,E1 -10047.492,E2 -10047.492} C_VEL
LIN {X 0,Y 418.322,Z 805.306,A -85,B 0,C 180,E1 -10048.963,E2 -10048.963} C_VEL
LIN {X 0,Y 418.195,Z 807.322,A -85,B 0,C 180,E1 -10050.832,E2 -10050.832} C_VEL
LIN {X 0,Y 418.201,Z 807.813,A -85,B 0,C 180,E1 -10051.93,E2 -10051.93} C_VEL
LIN {X 0,Y 418.217,Z 807.798,A -85,B 0,C 180,E1 -10053.017,E2 -10053.017} C_VEL
LIN {X 0,Y 418.325,Z 807.252,A -85,B 0,C 180,E1 -10054.099,E2 -10054.099} C_VEL
LIN {X 0,Y 418.472,Z 806.253,A -85,B 0,C 180,E1 -10055.174,E2 -10055.174} C_VEL
LIN {X 0,Y 418.733,Z 803.776,A -85,B 0,C 180,E1 -10056.77,E2 -10056.77} C_VEL
LIN {X 0,Y 419.04,Z 800.147,A -85,B 0,C 180,E1 -10058.347,E2 -10058.347} C_VEL
LIN {X 0,Y 419.564,Z 794.584,A -85,B 0,C 180,E1 -10060.102,E2 -10060.102} C_VEL
LIN {X 0,Y 420.05,Z 788.986,A -85,B 0,C 180,E1 -10061.464,E2 -10061.464} C_VEL
LIN {X 0,Y 420.743,Z 781.001,A -85,B 0,C 180,E1 -10063.003,E2 -10063.003} C_VEL
LIN {X 0,Y 421.371,Z 772.815,A -85,B 0,C 180,E1 -10064.274,E2 -10064.274} C_VEL
LIN {X 0,Y 422.055,Z 762.819,A -85,B 0,C 180,E1 -10065.535,E2 -10065.535} C_VEL
LIN {X 0,Y 422.668,Z 752.87,A -85,B 0,C 180,E1 -10066.539,E2 -10066.539} C_VEL
LIN {X 0,Y 423.116,Z 742.235,A -85,B 0,C 180,E1 -10067.408,E2 -10067.408} C_VEL
LIN {X 0,Y 422.939,Z 739.109,A -85,B 0,C 180,E1 -10067.646,E2 -10067.646} C_VEL
LIN {X 0,Y 419.412,Z 727.858,A -85,B 0,C 180,E1 -10068.522,E2 -10068.522} C_VEL
LIN {X 0,Y 418.335,Z 724.38,A -85,B 0,C 180,E1 -10068.768,E2 -10068.768} C_VEL
LIN {X 0,Y 418.415,Z 724.363,A -85,B 0,C 180,E1 -10072.313,E2 -10072.313} C_VEL
LIN {X 0,Y 418.498,Z 724.352,A -85,B 0,C 180,E1 -10074.217,E2 -10074.217} C_VEL
LIN {X 0,Y 418.544,Z 724.352,A -85,B 0,C 180,E1 -10078.075,E2 -10078.075} C_VEL
LIN {X 0,Y 418.671,Z 724.335,A -85,B 0,C 180,E1 -10080,E2 -10080} C_VEL
LIN {X 0,Y 418.497,Z 724.348,A -85,B 0,C 180,E1 -10082.888,E2 -10082.888} C_VEL
LIN {X 0,Y 418.512,Z 724.351,A -85,B 0,C 180,E1 -10085.783,E2 -10085.783} C_VEL
LIN {X 0,Y 418.399,Z 724.36,A -85,B 0,C 180,E1 -10088.695,E2 -10088.695} C_VEL
LIN {X 0,Y 418.318,Z 724.376,A -85,B 0,C 180,E1 -10091.631,E2 -10091.631} C_VEL
LIN {X 0,Y 418.307,Z 724.373,A -85,B 0,C 180,E1 -10094.597,E2 -10094.597} C_VEL
LIN {X 0,Y 418.29,Z 724.38,A -85,B 0,C 180,E1 -10097.604,E2 -10097.604} C_VEL
LIN {X 0,Y 418.254,Z 724.381,A -85,B 0,C 180,E1 -10100.663,E2 -10100.663} C_VEL
LIN {X 0,Y 418.278,Z 724.38,A -85,B 0,C 180,E1 -10103.782,E2 -10103.782} C_VEL
LIN {X 0,Y 418.313,Z 724.376,A -85,B 0,C 180,E1 -10107.07,E2 -10107.07} C_VEL
LIN {X 0,Y 418.248,Z 724.389,A -85,B 0,C 180,E1 -10110.272,E2 -10110.272} C_VEL
LIN {X 0,Y 418.252,Z 724.384,A -85,B 0,C 180,E1 -10113.677,E2 -10113.677} C_VEL
LIN {X 0,Y 418.243,Z 724.389,A -85,B 0,C 180,E1 -10117.224,E2 -10117.224} C_VEL
LIN {X 0,Y 418.254,Z 724.389,A -85,B 0,C 180,E1 -10119.682,E2 -10119.682} C_VEL
LIN {X 0,Y 418.233,Z 724.392,A -85,B 0,C 180,E1 -10122.321,E2 -10122.321} C_VEL
LIN {X 0,Y 418.238,Z 724.389,A -85,B 0,C 180,E1 -10125.109,E2 -10125.109} C_VEL
LIN {X 0,Y 418.243,Z 724.478,A -85,B 0,C 180,E1 -10126.854,E2 -10126.854} C_VEL
LIN {X 0,Y 419.585,Z 730.682,A -85,B 0,C 180,E1 -10129.213,E2 -10129.213} C_VEL
LIN {X 0,Y 421.031,Z 738.298,A -85,B 0,C 180,E1 -10131.857,E2 -10131.857} C_VEL
LIN {X 0,Y 421.546,Z 742.309,A -85,B 0,C 180,E1 -10133.155,E2 -10133.155} C_VEL
LIN {X 0,Y 420.853,Z 751.908,A -85,B 0,C 180,E1 -10135.983,E2 -10135.983} C_VEL
LIN {X 0,Y 420.197,Z 761.822,A -85,B 0,C 180,E1 -10138.769,E2 -10138.769} C_VEL
LIN {X 0,Y 419.457,Z 775.212,A -85,B 0,C 180,E1 -10142.38,E2 -10142.38} C_VEL
LIN {X 0,Y 418.877,Z 788.098,A -85,B 0,C 180,E1 -10145.728,E2 -10145.728} C_VEL
LIN {X 0,Y 418.407,Z 801.34,A -85,B 0,C 180,E1 -10149.088,E2 -10149.088} C_VEL
LIN {X 0,Y 418.056,Z 814.613,A -85,B 0,C 180,E1 -10152.386,E2 -10152.386} C_VEL
LIN {X 0,Y 418.022,Z 815.403,A -85,B 0,C 180,E1 -10152.58,E2 -10152.58} C_VEL
LIN {X 0,Y 419.596,Z 830.617,A -85,B 0,C 180,E1 -10153.099,E2 -10153.099} C_VEL
LIN {X 0,Y 420.358,Z 844.048,A -85,B 0,C 180,E1 -10153.737,E2 -10153.737} C_VEL
LIN {X 0,Y 421.039,Z 852.57,A -85,B 0,C 180,E1 -10154.261,E2 -10154.261} C_VEL
LIN {X 0,Y 420.24,Z 864.495,A -85,B 0,C 180,E1 -10155.1,E2 -10155.1} C_VEL
LIN {X 0,Y 419.499,Z 876.553,A -85,B 0,C 180,E1 -10156.188,E2 -10156.188} C_VEL
LIN {X 0,Y 419.005,Z 885.721,A -85,B 0,C 180,E1 -10157.203,E2 -10157.203} C_VEL
LIN {X 0,Y 418.43,Z 894.541,A -85,B 0,C 180,E1 -10158.372,E2 -10158.372} C_VEL
LIN {X 0,Y 417.939,Z 903.566,A -85,B 0,C 180,E1 -10159.83,E2 -10159.83} C_VEL
LIN {X 0,Y 417.672,Z 910.829,A -85,B 0,C 180,E1 -10161.289,E2 -10161.289} C_VEL
LIN {X 0,Y 417.548,Z 916.693,A -85,B 0,C 180,E1 -10162.748,E2 -10162.748} C_VEL
LIN {X 0,Y 417.514,Z 921.327,A -85,B 0,C 180,E1 -10164.203,E2 -10164.203} C_VEL
LIN {X 0,Y 417.568,Z 924.851,A -85,B 0,C 180,E1 -10165.656,E2 -10165.656} C_VEL
LIN {X 0,Y 417.541,Z 927.332,A -85,B 0,C 180,E1 -10167.105,E2 -10167.105} C_VEL
LIN {X 0,Y 417.549,Z 928.438,A -85,B 0,C 180,E1 -10168.071,E2 -10168.071} C_VEL
LIN {X 0,Y 417.542,Z 929.134,A -85,B 0,C 180,E1 -10169.035,E2 -10169.035} C_VEL
LIN {X 0,Y 417.543,Z 929.405,A -85,B 0,C 180,E1 -10170,E2 -10170} C_VEL
LIN {X 0,Y 417.531,Z 929.224,A -85,B 0,C 180,E1 -10170.964,E2 -10170.964} C_VEL
LIN {X 0,Y 417.526,Z 928.639,A -85,B 0,C 180,E1 -10171.929,E2 -10171.929} C_VEL
LIN {X 0,Y 417.518,Z 927.645,A -85,B 0,C 180,E1 -10172.894,E2 -10172.894} C_VEL
LIN {X 0,Y 417.59,Z 926.222,A -85,B 0,C 180,E1 -10173.86,E2 -10173.86} C_VEL
LIN {X 0,Y 417.464,Z 923.198,A -85,B 0,C 180,E1 -10175.313,E2 -10175.313} C_VEL
LIN {X 0,Y 417.476,Z 919.1,A -85,B 0,C 180,E1 -10176.767,E2 -10176.767} C_VEL
LIN {X 0,Y 417.637,Z 912.784,A -85,B 0,C 180,E1 -10178.467,E2 -10178.467} C_VEL
LIN {X 0,Y 417.862,Z 905.897,A -85,B 0,C 180,E1 -10179.927,E2 -10179.927} C_VEL
LIN {X 0,Y 418.317,Z 897.36,A -85,B 0,C 180,E1 -10181.385,E2 -10181.385} C_VEL
LIN {X 0,Y 418.926,Z 888.604,A -85,B 0,C 180,E1 -10182.597,E2 -10182.597} C_VEL
LIN {X 0,Y 419.549,Z 878.09,A -85,B 0,C 180,E1 -10183.785,E2 -10183.785} C_VEL
LIN {X 0,Y 420.168,Z 867.226,A -85,B 0,C 180,E1 -10184.778,E2 -10184.778} C_VEL
LIN {X 0,Y 420.998,Z 855.505,A -85,B 0,C 180,E1 -10185.616,E2 -10185.616} C_VEL
LIN {X 0,Y 420.961,Z 849.3,A -85,B 0,C 180,E1 -10185.99,E2 -10185.99} C_VEL
LIN {X 0,Y 419.799,Z 836.418,A -85,B 0,C 180,E1 -10186.648,E2 -10186.648} C_VEL
LIN {X 0,Y 418.558,Z 823.792,A -85,B 0,C 180,E1 -10187.112,E2 -10187.112} C_VEL
LIN {X 0,Y 418.033,Z 818.883,A -85,B 0,C 180,E1 -10187.254,E2 -10187.254} C_VEL
LIN {X 0,Y 418.523,Z 805.641,A -85,B 0,C 180,E1 -10190.649,E2 -10190.649} C_VEL
LIN {X 0,Y 419.038,Z 793.768,A -85,B 0,C 180,E1 -10193.736,E2 -10193.736} C_VEL
LIN {X 0,Y 419.798,Z 780.711,A -85,B 0,C 180,E1 -10197.181,E2 -10197.181} C_VEL
LIN {X 0,Y 420.579,Z 767.893,A -85,B 0,C 180,E1 -10200.642,E2 -10200.642} C_VEL
LIN {X 0,Y 421.487,Z 755.913,A -85,B 0,C 180,E1 -10203.958,E2 -10203.958} C_VEL
LIN {X 0,Y 422.305,Z 745.309,A -85,B 0,C 180,E1 -10206.983,E2 -10206.983} C_VEL
LIN {X 0,Y 421.264,Z 739.335,A -85,B 0,C 180,E1 -10208.834,E2 -10208.834} C_VEL
LIN {X 0,Y 419.519,Z 730.541,A -85,B 0,C 180,E1 -10211.689,E2 -10211.689} C_VEL
LIN {X 0,Y 418.229,Z 724.39,A -85,B 0,C 180,E1 -10213.809,E2 -10213.809} C_VEL
LIN {X 0,Y 418.21,Z 724.389,A -85,B 0,C 180,E1 -10216.449,E2 -10216.449} C_VEL
LIN {X 0,Y 418.225,Z 724.39,A -85,B 0,C 180,E1 -10219.13,E2 -10219.13} C_VEL
LIN {X 0,Y 418.23,Z 724.386,A -85,B 0,C 180,E1 -10222.167,E2 -10222.167} C_VEL
LIN {X 0,Y 418.267,Z 724.385,A -85,B 0,C 180,E1 -10225.42,E2 -10225.42} C_VEL
LIN {X 0,Y 418.213,Z 724.388,A -85,B 0,C 180,E1 -10228.604,E2 -10228.604} C_VEL
LIN {X 0,Y 418.293,Z 724.382,A -85,B 0,C 180,E1 -10231.937,E2 -10231.937} C_VEL
LIN {X 0,Y 418.292,Z 724.378,A -85,B 0,C 180,E1 -10235.163,E2 -10235.163} C_VEL
LIN {X 0,Y 418.236,Z 724.387,A -85,B 0,C 180,E1 -10238.304,E2 -10238.304} C_VEL
LIN {X 0,Y 418.283,Z 724.38,A -85,B 0,C 180,E1 -10241.383,E2 -10241.383} C_VEL
LIN {X 0,Y 418.304,Z 724.379,A -85,B 0,C 180,E1 -10244.406,E2 -10244.406} C_VEL
LIN {X 0,Y 418.358,Z 724.37,A -85,B 0,C 180,E1 -10247.386,E2 -10247.386} C_VEL
LIN {X 0,Y 418.402,Z 724.365,A -85,B 0,C 180,E1 -10251.305,E2 -10251.305} C_VEL
LIN {X 0,Y 418.512,Z 724.356,A -85,B 0,C 180,E1 -10254.217,E2 -10254.217} C_VEL
LIN {X 0,Y 418.541,Z 724.35,A -85,B 0,C 180,E1 -10258.076,E2 -10258.076} C_VEL
LIN {X 0,Y 418.669,Z 724.333,A -85,B 0,C 180,E1 -10260,E2 -10260} C_VEL
LIN {X 0,Y 418.495,Z 724.355,A -85,B 0,C 180,E1 -10262.888,E2 -10262.888} C_VEL
LIN {X 0,Y 418.459,Z 724.359,A -85,B 0,C 180,E1 -10266.529,E2 -10266.529} C_VEL
LIN {X 0,Y 418.341,Z 724.374,A -85,B 0,C 180,E1 -10269.672,E2 -10269.672} C_VEL
LIN {X 0,Y 418.349,Z 724.374,A -85,B 0,C 180,E1 -10273.001,E2 -10273.001} C_VEL
LIN {X 0,Y 418.315,Z 724.38,A -85,B 0,C 180,E1 -10276.735,E2 -10276.735} C_VEL
LIN {X 0,Y 418.273,Z 724.383,A -85,B 0,C 180,E1 -10279.79,E2 -10279.79} C_VEL
LIN {X 0,Y 418.229,Z 724.389,A -85,B 0,C 180,E1 -10282.737,E2 -10282.737} C_VEL
LIN {X 0,Y 418.231,Z 724.389,A -85,B 0,C 180,E1 -10285.907,E2 -10285.907} C_VEL
LIN {X 0,Y 418.262,Z 724.386,A -85,B 0,C 180,E1 -10289.162,E2 -10289.162} C_VEL
LIN {X 0,Y 418.253,Z 724.385,A -85,B 0,C 180,E1 -10292.843,E2 -10292.843} C_VEL
LIN {X 0,Y 418.244,Z 724.387,A -85,B 0,C 180,E1 -10296.237,E2 -10296.237} C_VEL
LIN {X 0,Y 418.2,Z 724.392,A -85,B 0,C 180,E1 -10299.688,E2 -10299.688} C_VEL
LIN {X 0,Y 418.21,Z 724.392,A -85,B 0,C 180,E1 -10302.318,E2 -10302.318} C_VEL
LIN {X 0,Y 418.236,Z 724.387,A -85,B 0,C 180,E1 -10305.109,E2 -10305.109} C_VEL
LIN {X 0,Y 418.22,Z 724.389,A -85,B 0,C 180,E1 -10307.764,E2 -10307.764} C_VEL
LIN {X 0,Y 418.235,Z 724.389,A -85,B 0,C 180,E1 -10311.556,E2 -10311.556} C_VEL
LIN {X 0,Y 418.25,Z 724.385,A -85,B 0,C 180,E1 -10315.158,E2 -10315.158} C_VEL
LIN {X 0,Y 418.232,Z 724.388,A -85,B 0,C 180,E1 -10317.471,E2 -10317.471} C_VEL
LIN {X 0,Y 418.261,Z 724.385,A -85,B 0,C 180,E1 -10320.898,E2 -10320.898} C_VEL
LIN {X 0,Y 418.212,Z 724.39,A -85,B 0,C 180,E1 -10324.092,E2 -10324.092} C_VEL
LIN {X 0,Y 418.229,Z 724.388,A -85,B 0,C 180,E1 -10327.263,E2 -10327.263} C_VEL
LIN {X 0,Y 418.286,Z 724.381,A -85,B 0,C 180,E1 -10330.364,E2 -10330.364} C_VEL
LIN {X 0,Y 418.318,Z 724.377,A -85,B 0,C 180,E1 -10333.405,E2 -10333.405} C_VEL
LIN {X 0,Y 418.349,Z 724.375,A -85,B 0,C 180,E1 -10337,E2 -10337} C_VEL
LIN {X 0,Y 418.322,Z 724.376,A -85,B 0,C 180,E1 -10340.328,E2 -10340.328} C_VEL
LIN {X 0,Y 418.444,Z 724.364,A -85,B 0,C 180,E1 -10343.248,E2 -10343.248} C_VEL
LIN {X 0,Y 418.316,Z 724.379,A -85,B 0,C 180,E1 -10345.181,E2 -10345.181} C_VEL
LIN {X 0,Y 418.536,Z 724.349,A -85,B 0,C 180,E1 -10348.076,E2 -10348.076} C_VEL
LIN {X 0,Y 418.409,Z 724.365,A -85,B 0,C 180,E1 -10350.963,E2 -10350.963} C_VEL
LIN {X 0,Y 418.474,Z 724.357,A -85,B 0,C 180,E1 -10352.888,E2 -10352.888} C_VEL
LIN {X 0,Y 418.487,Z 724.357,A -85,B 0,C 180,E1 -10355.783,E2 -10355.783} C_VEL
LIN {X 0,Y 418.379,Z 724.368,A -85,B 0,C 180,E1 -10358.696,E2 -10358.696} C_VEL
LIN {X 0,Y 418.318,Z 724.38,A -85,B 0,C 180,E1 -10361.631,E2 -10361.631} C_VEL
LIN {X 0,Y 418.327,Z 724.376,A -85,B 0,C 180,E1 -10363.317,E2 -10363.317} C_VEL
LIN {X 0,Y 417.632,Z 724.465,A -85,B 0,C 180,E1 -10364.121,E2 -10364.121} C_VEL
LIN {X 0,Y 414.755,Z 724.821,A -85,B 0,C 180,E1 -10365.426,E2 -10365.426} C_VEL
LIN {X 0,Y 412.342,Z 725.119,A -85,B 0,C 180,E1 -10366.48,E2 -10366.48} C_VEL
LIN {X 0,Y 411.319,Z 725.248,A -85,B 0,C 180,E1 -10367.295,E2 -10367.295} C_VEL
LIN {X 0,Y 411.241,Z 725.258,A -85,B 0,C 180,E1 -10367.571,E2 -10367.571} C_VEL
LIN {X 0,Y 411.2,Z 725.262,A -85,B 0,C 180,E1 -10371.034,E2 -10371.034} C_VEL
LIN {X 0,Y 411.207,Z 725.263,A -85,B 0,C 180,E1 -10374.217,E2 -10374.217} C_VEL
LIN {X 0,Y 411.192,Z 725.263,A -85,B 0,C 180,E1 -10377.483,E2 -10377.483} C_VEL
LIN {X 0,Y 411.192,Z 725.262,A -85,B 0,C 180,E1 -10380.848,E2 -10380.848} C_VEL
LIN {X 0,Y 411.208,Z 725.265,A -85,B 0,C 180,E1 -10384.334,E2 -10384.334} C_VEL
LIN {X 0,Y 411.195,Z 725.264,A -85,B 0,C 180,E1 -10387.974,E2 -10387.974} C_VEL
LIN {X 0,Y 411.167,Z 725.264,A -85,B 0,C 180,E1 -10391.228,E2 -10391.228} C_VEL
LIN {X 0,Y 411.179,Z 725.27,A -85,B 0,C 180,E1 -10394.49,E2 -10394.49} C_VEL
LIN {X 0,Y 411.226,Z 725.259,A -85,B 0,C 180,E1 -10395.659,E2 -10395.659} C_VEL
LIN {X 0,Y 414.762,Z 737.855,A -85,B 0,C 180,E1 -10396.594,E2 -10396.594} C_VEL
LIN {X 0,Y 415.285,Z 740.428,A -85,B 0,C 180,E1 -10396.803,E2 -10396.803} C_VEL
LIN {X 0,Y 414.726,Z 751.784,A -85,B 0,C 180,E1 -10397.732,E2 -10397.732} C_VEL
LIN {X 0,Y 414.105,Z 762.881,A -85,B 0,C 180,E1 -10398.879,E2 -10398.879} C_VEL
LIN {X 0,Y 413.532,Z 772.694,A -85,B 0,C 180,E1 -10400.132,E2 -10400.132} C_VEL
LIN {X 0,Y 412.896,Z 781.551,A -85,B 0,C 180,E1 -10401.534,E2 -10401.534} C_VEL
LIN {X 0,Y 412.398,Z 789.233,A -85,B 0,C 180,E1 -10403.044,E2 -10403.044} C_VEL
LIN {X 0,Y 411.971,Z 795.374,A -85,B 0,C 180,E1 -10404.548,E2 -10404.548} C_VEL
LIN {X 0,Y 411.674,Z 799.191,A -85,B 0,C 180,E1 -10405.711,E2 -10405.711} C_VEL
LIN {X 0,Y 411.479,Z 803.653,A -85,B 0,C 180,E1 -10407.451,E2 -10407.451} C_VEL
LIN {X 0,Y 411.272,Z 806.652,A -85,B 0,C 180,E1 -10409.159,E2 -10409.159} C_VEL
LIN {X 0,Y 411.186,Z 808.254,A -85,B 0,C 180,E1 -10410.657,E2 -10410.657} C_VEL
LIN {X 0,Y 411.2,Z 808.911,A -85,B 0,C 180,E1 -10412.518,E2 -10412.518} C_VEL
LIN {X 0,Y 411.254,Z 808.663,A -85,B 0,C 180,E1 -10413.62,E2 -10413.62} C_VEL
LIN {X 0,Y 411.436,Z 807.713,A -85,B 0,C 180,E1 -10414.868,E2 -10414.868} C_VEL
LIN {X 0,Y 411.562,Z 806.599,A -85,B 0,C 180,E1 -10415.805,E2 -10415.805} C_VEL
LIN {X 0,Y 411.82,Z 804.297,A -85,B 0,C 180,E1 -10417.154,E2 -10417.154} C_VEL
LIN {X 0,Y 412.295,Z 799.724,A -85,B 0,C 180,E1 -10419.024,E2 -10419.024} C_VEL
LIN {X 0,Y 412.788,Z 794.38,A -85,B 0,C 180,E1 -10420.61,E2 -10420.61} C_VEL
LIN {X 0,Y 413.402,Z 787.59,A -85,B 0,C 180,E1 -10422.181,E2 -10422.181} C_VEL
LIN {X 0,Y 414.06,Z 780.571,A -85,B 0,C 180,E1 -10423.483,E2 -10423.483} C_VEL
LIN {X 0,Y 414.698,Z 772.282,A -85,B 0,C 180,E1 -10424.746,E2 -10424.746} C_VEL
LIN {X 0,Y 415.373,Z 762.735,A -85,B 0,C 180,E1 -10425.923,E2 -10425.923} C_VEL
LIN {X 0,Y 416.05,Z 751.193,A -85,B 0,C 180,E1 -10427.066,E2 -10427.066} C_VEL
LIN {X 0,Y 416.424,Z 741.684,A -85,B 0,C 180,E1 -10427.821,E2 -10427.821} C_VEL
LIN {X 0,Y 413.1,Z 730.754,A -85,B 0,C 180,E1 -10428.717,E2 -10428.717} C_VEL
LIN {X 0,Y 411.286,Z 725.257,A -85,B 0,C 180,E1 -10429.135,E2 -10429.135} C_VEL
LIN {X 0,Y 411.375,Z 725.241,A -85,B 0,C 180,E1 -10432.26,E2 -10432.26} C_VEL
LIN {X 0,Y 411.443,Z 725.232,A -85,B 0,C 180,E1 -10434.117,E2 -10434.117} C_VEL
LIN {X 0,Y 411.513,Z 725.228,A -85,B 0,C 180,E1 -10438.042,E2 -10438.042} C_VEL
LIN {X 0,Y 411.64,Z 725.211,A -85,B 0,C 180,E1 -10440,E2 -10440} C_VEL
LIN {X 0,Y 411.454,Z 725.226,A -85,B 0,C 180,E1 -10442.937,E2 -10442.937} C_VEL
LIN {X 0,Y 411.473,Z 725.227,A -85,B 0,C 180,E1 -10445.882,E2 -10445.882} C_VEL
LIN {X 0,Y 411.336,Z 725.239,A -85,B 0,C 180,E1 -10448.846,E2 -10448.846} C_VEL
LIN {X 0,Y 411.287,Z 725.25,A -85,B 0,C 180,E1 -10451.833,E2 -10451.833} C_VEL
LIN {X 0,Y 411.264,Z 725.249,A -85,B 0,C 180,E1 -10454.852,E2 -10454.852} C_VEL
LIN {X 0,Y 411.255,Z 725.255,A -85,B 0,C 180,E1 -10457.915,E2 -10457.915} C_VEL
LIN {X 0,Y 411.2,Z 725.258,A -85,B 0,C 180,E1 -10461.034,E2 -10461.034} C_VEL
LIN {X 0,Y 411.223,Z 725.259,A -85,B 0,C 180,E1 -10464.216,E2 -10464.216} C_VEL
LIN {X 0,Y 411.262,Z 725.255,A -85,B 0,C 180,E1 -10467.477,E2 -10467.477} C_VEL
LIN {X 0,Y 411.192,Z 725.263,A -85,B 0,C 180,E1 -10470.847,E2 -10470.847} C_VEL
LIN {X 0,Y 411.209,Z 725.267,A -85,B 0,C 180,E1 -10474.333,E2 -10474.333} C_VEL
LIN {X 0,Y 411.199,Z 725.268,A -85,B 0,C 180,E1 -10477.973,E2 -10477.973} C_VEL
LIN {X 0,Y 411.185,Z 725.27,A -85,B 0,C 180,E1 -10480.504,E2 -10480.504} C_VEL
LIN {X 0,Y 411.176,Z 725.269,A -85,B 0,C 180,E1 -10483.133,E2 -10483.133} C_VEL
LIN {X 0,Y 411.181,Z 725.377,A -85,B 0,C 180,E1 -10486.412,E2 -10486.412} C_VEL
LIN {X 0,Y 412.71,Z 732.355,A -85,B 0,C 180,E1 -10489.138,E2 -10489.138} C_VEL
LIN {X 0,Y 414.159,Z 740.048,A -85,B 0,C 180,E1 -10491.869,E2 -10491.869} C_VEL
LIN {X 0,Y 414.594,Z 744.163,A -85,B 0,C 180,E1 -10493.223,E2 -10493.223} C_VEL
LIN {X 0,Y 413.747,Z 754.581,A -85,B 0,C 180,E1 -10496.338,E2 -10496.338} C_VEL
LIN {X 0,Y 413.163,Z 763.061,A -85,B 0,C 180,E1 -10498.769,E2 -10498.769} C_VEL
LIN {X 0,Y 412.401,Z 776.245,A -85,B 0,C 180,E1 -10502.396,E2 -10502.396} C_VEL
LIN {X 0,Y 411.788,Z 789.148,A -85,B 0,C 180,E1 -10505.819,E2 -10505.819} C_VEL
LIN {X 0,Y 411.286,Z 802.36,A -85,B 0,C 180,E1 -10509.233,E2 -10509.233} C_VEL
LIN {X 0,Y 410.981,Z 814.127,A -85,B 0,C 180,E1 -10512.222,E2 -10512.222} C_VEL
LIN {X 0,Y 412.691,Z 830.531,A -85,B 0,C 180,E1 -10512.819,E2 -10512.819} C_VEL
LIN {X 0,Y 413.382,Z 843.347,A -85,B 0,C 180,E1 -10513.455,E2 -10513.455} C_VEL
LIN {X 0,Y 414.05,Z 853.699,A -85,B 0,C 180,E1 -10514.115,E2 -10514.115} C_VEL
LIN {X 0,Y 413.246,Z 865.059,A -85,B 0,C 180,E1 -10514.968,E2 -10514.968} C_VEL
LIN {X 0,Y 412.508,Z 875.581,A -85,B 0,C 180,E1 -10515.949,E2 -10515.949} C_VEL
LIN {X 0,Y 411.972,Z 884.916,A -85,B 0,C 180,E1 -10517.007,E2 -10517.007} C_VEL
LIN {X 0,Y 411.395,Z 893.494,A -85,B 0,C 180,E1 -10518.17,E2 -10518.17} C_VEL
LIN {X 0,Y 410.863,Z 902.512,A -85,B 0,C 180,E1 -10519.653,E2 -10519.653} C_VEL
LIN {X 0,Y 410.601,Z 909.783,A -85,B 0,C 180,E1 -10521.138,E2 -10521.138} C_VEL
LIN {X 0,Y 410.475,Z 915.654,A -85,B 0,C 180,E1 -10522.622,E2 -10522.622} C_VEL
LIN {X 0,Y 410.458,Z 920.295,A -85,B 0,C 180,E1 -10524.103,E2 -10524.103} C_VEL
LIN {X 0,Y 410.529,Z 923.826,A -85,B 0,C 180,E1 -10525.582,E2 -10525.582} C_VEL
LIN {X 0,Y 410.502,Z 926.31,A -85,B 0,C 180,E1 -10527.056,E2 -10527.056} C_VEL
LIN {X 0,Y 410.513,Z 927.418,A -85,B 0,C 180,E1 -10528.038,E2 -10528.038} C_VEL
LIN {X 0,Y 410.512,Z 928.118,A -85,B 0,C 180,E1 -10529.019,E2 -10529.019} C_VEL
LIN {X 0,Y 410.517,Z 928.386,A -85,B 0,C 180,E1 -10530,E2 -10530} C_VEL
LIN {X 0,Y 410.501,Z 928.203,A -85,B 0,C 180,E1 -10530.981,E2 -10530.981} C_VEL
LIN {X 0,Y 410.491,Z 927.616,A -85,B 0,C 180,E1 -10531.962,E2 -10531.962} C_VEL
LIN {X 0,Y 410.481,Z 926.622,A -85,B 0,C 180,E1 -10532.944,E2 -10532.944} C_VEL
LIN {X 0,Y 410.556,Z 925.188,A -85,B 0,C 180,E1 -10533.926,E2 -10533.926} C_VEL
LIN {X 0,Y 410.421,Z 922.152,A -85,B 0,C 180,E1 -10535.404,E2 -10535.404} C_VEL
LIN {X 0,Y 410.425,Z 918.036,A -85,B 0,C 180,E1 -10536.884,E2 -10536.884} C_VEL
LIN {X 0,Y 410.591,Z 911.7,A -85,B 0,C 180,E1 -10538.614,E2 -10538.614} C_VEL
LIN {X 0,Y 410.792,Z 904.789,A -85,B 0,C 180,E1 -10540.1,E2 -10540.1} C_VEL
LIN {X 0,Y 411.309,Z 896.224,A -85,B 0,C 180,E1 -10541.582,E2 -10541.582} C_VEL
LIN {X 0,Y 411.975,Z 887.446,A -85,B 0,C 180,E1 -10542.813,E2 -10542.813} C_VEL
LIN {X 0,Y 412.517,Z 877.832,A -85,B 0,C 180,E1 -10543.925,E2 -10543.925} C_VEL
LIN {X 0,Y 413.25,Z 865.988,A -85,B 0,C 180,E1 -10545.032,E2 -10545.032} C_VEL
LIN {X 0,Y 414.099,Z 854.184,A -85,B 0,C 180,E1 -10545.883,E2 -10545.883} C_VEL
LIN {X 0,Y 413.552,Z 845.618,A -85,B 0,C 180,E1 -10546.411,E2 -10546.411} C_VEL
LIN {X 0,Y 412.532,Z 832.497,A -85,B 0,C 180,E1 -10547.041,E2 -10547.041} C_VEL
LIN {X 0,Y 410.987,Z 817.957,A -85,B 0,C 180,E1 -10547.538,E2 -10547.538} C_VEL
LIN {X 0,Y 411.571,Z 802.727,A -85,B 0,C 180,E1 -10551.539,E2 -10551.539} C_VEL
LIN {X 0,Y 412.185,Z 790.875,A -85,B 0,C 180,E1 -10554.692,E2 -10554.692} C_VEL
LIN {X 0,Y 413.027,Z 776.986,A -85,B 0,C 180,E1 -10558.453,E2 -10558.453} C_VEL
LIN {X 0,Y 414.006,Z 763.005,A -85,B 0,C 180,E1 -10562.339,E2 -10562.339} C_VEL
LIN {X 0,Y 414.982,Z 751.548,A -85,B 0,C 180,E1 -10565.618,E2 -10565.618} C_VEL
LIN {X 0,Y 415.289,Z 745.79,A -85,B 0,C 180,E1 -10567.308,E2 -10567.308} C_VEL
LIN {X 0,Y 413.526,Z 736.718,A -85,B 0,C 180,E1 -10570.227,E2 -10570.227} C_VEL
LIN {X 0,Y 411.569,Z 727.12,A -85,B 0,C 180,E1 -10573.47,E2 -10573.47} C_VEL
LIN {X 0,Y 411.188,Z 725.267,A -85,B 0,C 180,E1 -10574.122,E2 -10574.122} C_VEL
LIN {X 0,Y 411.183,Z 725.268,A -85,B 0,C 180,E1 -10577.304,E2 -10577.304} C_VEL
LIN {X 0,Y 411.219,Z 725.26,A -85,B 0,C 180,E1 -10580.776,E2 -10580.776} C_VEL
LIN {X 0,Y 411.2,Z 725.261,A -85,B 0,C 180,E1 -10584.471,E2 -10584.471} C_VEL
LIN {X 0,Y 411.209,Z 725.26,A -85,B 0,C 180,E1 -10586.873,E2 -10586.873} C_VEL
LIN {X 0,Y 411.235,Z 725.257,A -85,B 0,C 180,E1 -10590.644,E2 -10590.644} C_VEL
LIN {X 0,Y 411.239,Z 725.26,A -85,B 0,C 180,E1 -10593.619,E2 -10593.619} C_VEL
LIN {X 0,Y 411.198,Z 725.262,A -85,B 0,C 180,E1 -10596.852,E2 -10596.852} C_VEL
LIN {X 0,Y 411.217,Z 725.264,A -85,B 0,C 180,E1 -10600.05,E2 -10600.05} C_VEL
LIN {X 0,Y 411.265,Z 725.254,A -85,B 0,C 180,E1 -10603.131,E2 -10603.131} C_VEL
LIN {X 0,Y 411.308,Z 725.249,A -85,B 0,C 180,E1 -10606.896,E2 -10606.896} C_VEL
LIN {X 0,Y 411.294,Z 725.255,A -85,B 0,C 180,E1 -10610.161,E2 -10610.161} C_VEL
